C07286=1065.476,339.617,397.493,174.276,33.867,156.261
C07287=1065.483,339.864,397.457,174.280,33.872,156.262
C07288=1065.489,340.112,397.422,174.283,33.877,156.263
C07289=1065.496,340.359,397.387,174.287,33.882,156.264
C07290=1065.501,340.606,397.351,174.291,33.887,156.265
C07291=1065.508,340.853,397.316,174.295,33.893,156.266
C07292=1065.515,341.101,397.281,174.298,33.897,156.267
C07293=1065.521,341.348,397.245,174.302,33.902,156.268
C07294=1065.528,341.596,397.210,174.305,33.908,156.269
C07295=1065.535,341.843,397.175,174.310,33.912,156.270
C07296=1065.541,342.091,397.139,174.313,33.918,156.271
C07297=1065.547,342.338,397.104,174.317,33.923,156.272
C07298=1065.554,342.585,397.069,174.320,33.928,156.273
C07299=1065.560,342.833,397.033,174.324,33.933,156.274
C07300=1065.567,343.081,396.998,174.328,33.938,156.275
C07301=1065.574,343.327,396.962,174.332,33.943,156.276
C07302=1065.581,343.576,396.926,174.336,33.949,156.278
C07303=1065.587,343.823,396.891,174.339,33.954,156.279
C07304=1065.593,344.071,396.855,174.343,33.959,156.280
C07305=1065.601,344.317,396.820,174.347,33.964,156.281
C07306=1065.607,344.565,396.784,174.351,33.969,156.282
C07307=1065.612,344.796,396.751,174.354,33.974,156.283
C07308=1065.618,345.028,396.717,174.358,33.979,156.284
C07309=1065.625,345.260,396.684,174.361,33.984,156.285
C07310=1065.631,345.491,396.650,174.364,33.989,156.286
C07311=1065.637,345.724,396.617,174.369,33.994,156.287
C07312=1065.644,345.955,396.583,174.372,33.998,156.288
C07313=1065.649,346.186,396.550,174.375,34.004,156.289
C07314=1065.655,346.418,396.516,174.379,34.008,156.290
C07315=1065.661,346.665,396.480,174.383,34.013,156.291
C07316=1065.668,346.912,396.444,174.387,34.019,156.292
C07317=1065.675,347.161,396.409,174.390,34.024,156.293
C07318=1065.682,347.408,396.372,174.394,34.029,156.294
C07319=1065.689,347.654,396.336,174.398,34.035,156.296
C07320=1065.695,347.902,396.301,174.402,34.040,156.297
C07321=1065.701,348.149,396.264,174.406,34.045,156.298
C07322=1065.708,348.396,396.229,174.409,34.051,156.299
C07323=1065.714,348.643,396.192,174.413,34.056,156.300
C07324=1065.721,348.891,396.156,174.418,34.062,156.301
C07325=1065.727,349.139,396.120,174.421,34.067,156.302
C07326=1065.734,349.386,396.084,174.425,34.072,156.303
C07327=1065.740,349.633,396.048,174.429,34.077,156.304
C07328=1065.747,349.881,396.012,174.433,34.083,156.306
C07329=1065.754,350.128,395.976,174.437,34.088,156.307
C07330=1065.760,350.375,395.939,174.441,34.093,156.308
C07331=1065.767,350.622,395.903,174.444,34.099,156.309
C07332=1065.774,350.870,395.866,174.448,34.104,156.310
C07333=1065.781,351.117,395.831,174.453,34.110,156.311
C07334=1065.787,351.364,395.794,174.456,34.115,156.312
C07335=1065.793,351.611,395.758,174.460,34.121,156.314
C07336=1065.800,351.859,395.721,174.464,34.126,156.315
C07337=1065.807,352.106,395.685,174.468,34.131,156.316
C07338=1065.814,352.353,395.649,174.472,34.137,156.317
C07339=1065.820,352.600,395.612,174.476,34.142,156.318
C07340=1065.827,352.848,395.576,174.479,34.148,156.319
C07341=1065.833,353.095,395.539,174.484,34.153,156.321
C07342=1065.840,353.342,395.502,174.488,34.159,156.322
C07343=1065.846,353.589,395.466,174.491,34.164,156.323
C07344=1065.853,353.836,395.429,174.496,34.170,156.324
C07345=1065.860,354.084,395.393,174.500,34.175,156.325
C07346=1065.866,354.331,395.356,174.503,34.181,156.326
C07347=1065.872,354.578,395.320,174.507,34.187,156.328
C07348=1065.880,354.825,395.282,174.512,34.192,156.329
C07349=1065.886,355.072,395.246,174.516,34.198,156.330
C07350=1065.892,355.320,395.209,174.519,34.203,156.331
C07351=1065.899,355.567,395.173,174.523,34.209,156.332
C07352=1065.906,355.814,395.136,174.528,34.214,156.333
C07353=1065.913,356.061,395.099,174.532,34.220,156.335
C07354=1065.919,356.309,395.062,174.535,34.226,156.336
C07355=1065.926,356.556,395.025,174.540,34.232,156.337
C07356=1065.933,356.803,394.988,174.544,34.237,156.338
C07357=1065.939,357.050,394.952,174.548,34.243,156.339
C07358=1065.946,357.298,394.915,174.551,34.248,156.341
C07359=1065.953,357.544,394.878,174.556,34.254,156.342
C07360=1065.960,357.792,394.841,174.560,34.260,156.343
C07361=1065.966,358.038,394.804,174.564,34.265,156.344
C07362=1065.973,358.286,394.767,174.568,34.271,156.346
C07363=1065.979,358.520,394.732,174.572,34.276,156.347
C07364=1065.986,358.753,394.697,174.576,34.281,156.348
C07365=1065.992,358.987,394.662,174.579,34.287,156.349
C07366=1065.999,359.221,394.626,174.584,34.292,156.350
C07367=1066.005,359.454,394.591,174.587,34.298,156.351
C07368=1066.011,359.688,394.556,174.591,34.303,156.352
C07369=1066.017,359.922,394.521,174.596,34.309,156.354
C07370=1066.024,360.155,394.486,174.599,34.315,156.355
C07371=1066.030,360.402,394.449,174.603,34.320,156.356
C07372=1066.038,360.649,394.412,174.608,34.326,156.357
C07373=1066.044,360.896,394.374,174.612,34.332,156.359
C07374=1066.051,361.143,394.338,174.615,34.337,156.360
C07375=1066.058,361.391,394.300,174.620,34.343,156.361
C07376=1066.064,361.637,394.262,174.624,34.349,156.362
C07377=1066.071,361.885,394.225,174.628,34.355,156.364
C07378=1066.078,362.132,394.188,174.632,34.361,156.365
C07379=1066.084,362.379,394.150,174.637,34.367,156.366
C07380=1066.092,362.626,394.113,174.641,34.373,156.367
C07381=1066.098,362.873,394.076,174.644,34.379,156.369
C07382=1066.105,363.120,394.037,174.649,34.385,156.370
C07383=1066.112,363.367,394.000,174.653,34.391,156.371
C07384=1066.119,363.614,393.963,174.657,34.396,156.373
C07385=1066.126,363.861,393.925,174.662,34.403,156.374
C07386=1066.132,364.108,393.887,174.666,34.408,156.375
C07387=1066.139,364.355,393.850,174.671,34.414,156.377
C07388=1066.146,364.602,393.812,174.675,34.420,156.378
C07389=1066.153,364.849,393.774,174.678,34.426,156.379
C07390=1066.159,365.097,393.736,174.683,34.432,156.380
C07391=1066.166,365.343,393.699,174.687,34.438,156.382
C07392=1066.172,365.591,393.661,174.691,34.445,156.383
C07393=1066.180,365.838,393.623,174.696,34.451,156.384
C07394=1066.186,366.084,393.586,174.700,34.457,156.386
C07395=1066.193,366.331,393.547,174.704,34.463,156.387
C07396=1066.200,366.578,393.509,174.709,34.469,156.388
C07397=1066.207,366.825,393.472,174.713,34.475,156.390
C07398=1066.213,367.072,393.434,174.718,34.481,156.391
C07399=1066.220,367.319,393.396,174.722,34.487,156.392
C07400=1066.227,367.566,393.358,174.725,34.493,156.394
C07401=1066.233,367.814,393.320,174.730,34.500,156.395
C07402=1066.241,368.060,393.281,174.734,34.506,156.396
C07403=1066.247,368.307,393.244,174.738,34.512,156.398
C07404=1066.254,368.554,393.206,174.743,34.518,156.399
C07405=1066.261,368.801,393.167,174.747,34.524,156.400
C07406=1066.267,369.048,393.129,174.752,34.530,156.402
C07407=1066.275,369.295,393.091,174.756,34.536,156.403
C07408=1066.281,369.542,393.053,174.760,34.543,156.404
C07409=1066.289,369.789,393.014,174.765,34.549,156.406
C07410=1066.295,370.036,392.977,174.769,34.555,156.407
C07411=1066.302,370.282,392.938,174.774,34.562,156.409
C07412=1066.309,370.529,392.900,174.778,34.568,156.410
C07413=1066.316,370.776,392.861,174.782,34.574,156.411
C07414=1066.323,371.023,392.823,174.787,34.581,156.413
C07415=1066.330,371.270,392.785,174.791,34.587,156.414
C07416=1066.337,371.517,392.746,174.796,34.593,156.416
C07417=1066.344,371.764,392.708,174.800,34.599,156.417
C07418=1066.351,372.011,392.670,174.805,34.606,156.418
C07419=1066.358,372.254,392.632,174.809,34.612,156.420
C07420=1066.364,372.496,392.594,174.813,34.618,156.421
C07421=1066.371,372.737,392.556,174.818,34.625,156.423
C07422=1066.378,372.980,392.518,174.822,34.631,156.424
C07423=1066.385,373.222,392.480,174.827,34.637,156.425
C07424=1066.392,373.465,392.442,174.831,34.644,156.427
C07425=1066.398,373.707,392.405,174.836,34.650,156.428
C07426=1066.405,373.950,392.367,174.840,34.656,156.430
C07427=1066.412,374.197,392.328,174.844,34.663,156.431
C07428=1066.419,374.444,392.289,174.849,34.669,156.432
C07429=1066.426,374.690,392.250,174.853,34.676,156.434
C07430=1066.433,374.937,392.211,174.858,34.683,156.435
C07431=1066.439,375.184,392.173,174.862,34.689,156.437
C07432=1066.447,375.430,392.133,174.867,34.695,156.438
C07433=1066.453,375.677,392.094,174.872,34.702,156.440
C07434=1066.460,375.924,392.055,174.877,34.708,156.441
C07435=1066.467,376.171,392.017,174.881,34.715,156.443
C07436=1066.474,376.418,391.978,174.886,34.722,156.444
C07437=1066.481,376.664,391.939,174.890,34.729,156.446
C07438=1066.487,376.911,391.900,174.895,34.735,156.447
C07439=1066.495,377.158,391.860,174.899,34.742,156.449
C07440=1066.502,377.405,391.821,174.903,34.748,156.450
C07441=1066.509,377.652,391.782,174.908,34.755,156.452
C07442=1066.516,377.899,391.744,174.913,34.762,156.453
C07443=1066.523,378.145,391.704,174.918,34.768,156.455
C07444=1066.530,378.392,391.665,174.922,34.775,156.456
C07445=1066.537,378.639,391.625,174.927,34.782,156.458
C07446=1066.544,378.885,391.586,174.931,34.789,156.459
C07447=1066.551,379.132,391.548,174.936,34.795,156.461
C07448=1066.558,379.378,391.508,174.941,34.802,156.462
C07449=1066.565,379.626,391.469,174.946,34.809,156.464
C07450=1066.573,379.872,391.429,174.950,34.816,156.465
C07451=1066.579,380.119,391.391,174.955,34.823,156.467
C07452=1066.587,380.366,391.351,174.960,34.829,156.468
C07453=1066.594,380.613,391.312,174.965,34.836,156.470
C07454=1066.601,380.859,391.272,174.970,34.843,156.471
C07455=1066.609,381.106,391.232,174.974,34.850,156.473
C07456=1066.616,381.353,391.193,174.979,34.857,156.474
C07457=1066.622,381.599,391.153,174.983,34.864,156.476
C07458=1066.630,381.846,391.113,174.989,34.871,156.478
C07459=1066.636,382.093,391.075,174.993,34.878,156.479
C07460=1066.643,382.339,391.034,174.998,34.885,156.481
C07461=1066.651,382.586,390.994,175.002,34.892,156.482
C07462=1066.658,382.832,390.955,175.008,34.899,156.484
C07463=1066.664,383.079,390.915,175.012,34.906,156.485
C07464=1066.672,383.326,390.875,175.017,34.913,156.487
C07465=1066.679,383.573,390.836,175.022,34.920,156.489
C07466=1066.685,383.819,390.796,175.027,34.928,156.490
C07467=1066.693,384.066,390.756,175.032,34.934,156.492
C07468=1066.700,384.312,390.716,175.036,34.941,156.494
C07469=1066.707,384.560,390.676,175.041,34.949,156.495
C07470=1066.714,384.806,390.636,175.047,34.956,156.497
C07471=1066.720,385.052,390.596,175.051,34.963,156.498
C07472=1066.728,385.299,390.556,175.056,34.970,156.500
C07473=1066.735,385.545,390.516,175.061,34.978,156.502
C07474=1066.742,385.792,390.475,175.066,34.985,156.503
C07475=1066.750,386.060,390.432,175.072,34.993,156.505
C07476=1066.758,386.328,390.389,175.076,35.000,156.507
C07477=1066.766,386.596,390.345,175.082,35.008,156.509
C07478=1066.774,386.865,390.302,175.088,35.016,156.510
C07479=1066.782,387.111,390.261,175.092,35.024,156.512
C07480=1066.788,387.357,390.221,175.097,35.031,156.514
C07481=1066.796,387.604,390.181,175.102,35.038,156.516
C07482=1066.802,387.851,390.141,175.107,35.045,156.517
C07483=1066.810,388.097,390.100,175.113,35.052,156.519
C07484=1066.817,388.344,390.060,175.117,35.060,156.521
C07485=1066.825,388.590,390.019,175.122,35.067,156.522
C07486=1066.832,388.837,389.979,175.128,35.075,156.524
C07487=1066.840,389.083,389.938,175.132,35.082,156.526
C07488=1066.847,389.330,389.899,175.137,35.089,156.527
C07489=1066.854,389.576,389.857,175.143,35.097,156.529
C07490=1066.862,389.823,389.817,175.147,35.104,156.531
C07491=1066.868,390.069,389.777,175.153,35.112,156.533
C07492=1066.876,390.316,389.737,175.157,35.119,156.534
C07493=1066.884,390.563,389.695,175.163,35.127,156.536
C07494=1066.890,390.810,389.655,175.168,35.134,156.538
C07495=1066.898,391.055,389.615,175.174,35.142,156.539
C07496=1066.905,391.302,389.573,175.178,35.150,156.541
C07497=1066.912,391.549,389.532,175.183,35.157,156.543
C07498=1066.920,391.795,389.492,175.189,35.165,156.545
C07499=1066.927,392.041,389.451,175.193,35.173,156.547
C07500=1066.934,392.288,389.410,175.199,35.181,156.548
C07501=1066.942,392.534,389.370,175.204,35.188,156.550
C07502=1066.949,392.781,389.328,175.209,35.196,156.552
C07503=1066.956,393.027,389.287,175.214,35.204,156.554
C07504=1066.963,393.273,389.246,175.220,35.211,156.556
C07505=1066.971,393.520,389.206,175.225,35.219,156.557
C07506=1066.979,393.766,389.164,175.230,35.227,156.559
C07507=1066.986,394.013,389.123,175.235,35.234,156.561
C07508=1066.993,394.259,389.082,175.241,35.243,156.563
C07509=1067.000,394.505,389.041,175.246,35.250,156.565
C07510=1067.007,394.752,389.000,175.251,35.258,156.566
C07511=1067.015,394.998,388.959,175.256,35.266,156.568
C07512=1067.023,395.245,388.918,175.262,35.274,156.570
C07513=1067.030,395.491,388.877,175.267,35.282,156.572
C07514=1067.038,395.737,388.835,175.272,35.290,156.574
C07515=1067.045,395.984,388.794,175.278,35.298,156.576
C07516=1067.052,396.230,388.752,175.283,35.306,156.578
C07517=1067.059,396.477,388.711,175.289,35.314,156.579
C07518=1067.067,396.723,388.669,175.293,35.322,156.581
C07519=1067.074,396.970,388.628,175.299,35.330,156.583
C07520=1067.082,397.216,388.587,175.304,35.338,156.585
C07521=1067.089,397.462,388.545,175.310,35.346,156.587
C07522=1067.096,397.709,388.503,175.316,35.354,156.589
C07523=1067.104,397.955,388.462,175.320,35.362,156.591
C07524=1067.111,398.201,388.420,175.326,35.370,156.593
C07525=1067.119,398.447,388.378,175.332,35.379,156.595
C07526=1067.127,398.695,388.337,175.337,35.387,156.597
C07527=1067.134,398.941,388.295,175.343,35.395,156.598
C07528=1067.142,399.187,388.254,175.348,35.403,156.600
C07529=1067.149,399.433,388.211,175.353,35.412,156.602
C07530=1067.156,399.679,388.169,175.359,35.420,156.604
C07531=1067.165,399.963,388.121,175.365,35.429,156.607
C07532=1067.174,400.249,388.073,175.372,35.439,156.609
C07533=1067.182,400.533,388.025,175.378,35.449,156.611
C07534=1067.191,400.817,387.976,175.384,35.459,156.614
C07535=1067.198,401.064,387.933,175.390,35.467,156.615
C07536=1067.206,401.310,387.891,175.396,35.475,156.617
C07537=1067.214,401.556,387.850,175.401,35.484,156.619
C07538=1067.221,401.802,387.808,175.407,35.492,156.621
C07539=1067.229,402.048,387.765,175.413,35.501,156.623
C07540=1067.236,402.295,387.723,175.419,35.509,156.625
C07541=1067.244,402.541,387.681,175.423,35.517,156.627
C07542=1067.252,402.787,387.638,175.429,35.526,156.630
C07543=1067.260,403.033,387.597,175.435,35.535,156.632
C07544=1067.266,403.279,387.554,175.441,35.544,156.634
C07545=1067.275,403.526,387.512,175.446,35.552,156.636
C07546=1067.282,403.772,387.470,175.452,35.561,156.638
C07547=1067.290,404.019,387.427,175.458,35.570,156.640
C07548=1067.297,404.265,387.385,175.464,35.578,156.642
C07549=1067.304,404.511,387.342,175.470,35.587,156.644
C07550=1067.313,404.757,387.299,175.475,35.596,156.646
C07551=1067.320,405.003,387.257,175.481,35.604,156.648
C07552=1067.328,405.250,387.214,175.487,35.613,156.650
C07553=1067.336,405.496,387.172,175.493,35.622,156.652
C07554=1067.343,405.743,387.129,175.499,35.631,156.655
C07555=1067.351,405.988,387.086,175.505,35.640,156.657
C07556=1067.358,406.235,387.043,175.511,35.649,156.659
C07557=1067.366,406.480,387.001,175.516,35.657,156.661
C07558=1067.374,406.727,386.958,175.522,35.666,156.663
C07559=1067.381,406.973,386.915,175.528,35.676,156.665
C07560=1067.389,407.220,386.872,175.534,35.684,156.667
C07561=1067.396,407.465,386.829,175.540,35.694,156.670
C07562=1067.404,407.712,386.785,175.546,35.703,156.672
C07563=1067.412,407.958,386.743,175.552,35.712,156.674
C07564=1067.419,408.204,386.700,175.558,35.721,156.676
C07565=1067.427,408.450,386.656,175.564,35.730,156.678
C07566=1067.435,408.696,386.614,175.570,35.739,156.681
C07567=1067.443,408.943,386.571,175.576,35.749,156.683
C07568=1067.450,409.189,386.527,175.582,35.758,156.685
C07569=1067.458,409.435,386.484,175.588,35.767,156.687
C07570=1067.466,409.681,386.441,175.595,35.776,156.690
C07571=1067.474,409.927,386.397,175.601,35.785,156.692
C07572=1067.482,410.173,386.354,175.607,35.795,156.694
C07573=1067.489,410.419,386.311,175.613,35.804,156.696
C07574=1067.497,410.665,386.267,175.619,35.813,156.699
C07575=1067.505,410.912,386.224,175.625,35.823,156.701
C07576=1067.513,411.158,386.181,175.631,35.832,156.703
C07577=1067.521,411.403,386.137,175.637,35.842,156.705
C07578=1067.528,411.650,386.094,175.643,35.851,156.708
C07579=1067.537,411.896,386.051,175.650,35.860,156.710
C07580=1067.545,412.142,386.006,175.656,35.870,156.712
C07581=1067.553,412.388,385.963,175.662,35.879,156.715
C07582=1067.560,412.634,385.919,175.668,35.889,156.717
C07583=1067.569,412.880,385.876,175.674,35.898,156.719
C07584=1067.577,413.126,385.832,175.682,35.908,156.722
C07585=1067.585,413.373,385.788,175.688,35.918,156.724
C07586=1067.593,413.618,385.744,175.694,35.927,156.726
C07587=1067.601,413.907,385.693,175.701,35.939,156.729
C07588=1067.612,414.195,385.642,175.709,35.950,156.732
C07589=1067.621,414.484,385.590,175.716,35.961,156.735
C07590=1067.630,414.772,385.539,175.724,35.973,156.738
C07591=1067.638,415.018,385.494,175.731,35.982,156.740
C07592=1067.646,415.265,385.451,175.737,35.993,156.742
C07593=1067.654,415.510,385.406,175.743,36.002,156.745
C07594=1067.662,415.756,385.362,175.750,36.012,156.747
C07595=1067.670,416.002,385.318,175.756,36.022,156.750
C07596=1067.678,416.248,385.274,175.763,36.032,156.752
C07597=1067.686,416.494,385.230,175.770,36.042,156.755
C07598=1067.694,416.740,385.185,175.776,36.052,156.757
C07599=1067.703,416.986,385.141,175.783,36.062,156.760
C07600=1067.710,417.232,385.096,175.790,36.073,156.762
C07601=1067.718,417.478,385.051,175.796,36.083,156.765
C07602=1067.726,417.724,385.007,175.803,36.093,156.767
C07603=1067.734,417.969,384.963,175.810,36.103,156.770
C07604=1067.742,418.215,384.918,175.816,36.113,156.772
C07605=1067.751,418.462,384.874,175.823,36.123,156.775
C07606=1067.759,418.707,384.829,175.830,36.134,156.777
C07607=1067.767,418.953,384.785,175.836,36.144,156.780
C07608=1067.775,419.198,384.739,175.844,36.154,156.782
C07609=1067.783,419.445,384.695,175.850,36.165,156.785
C07610=1067.791,419.691,384.650,175.857,36.175,156.788
C07611=1067.800,419.936,384.606,175.864,36.185,156.790
C07612=1067.808,420.182,384.561,175.870,36.196,156.793
C07613=1067.817,420.428,384.516,175.878,36.206,156.795
C07614=1067.824,420.673,384.470,175.884,36.217,156.798
C07615=1067.833,420.920,384.426,175.892,36.227,156.801
C07616=1067.841,421.165,384.381,175.898,36.238,156.803
C07617=1067.849,421.411,384.336,175.906,36.248,156.806
C07618=1067.858,421.657,384.290,175.912,36.259,156.809
C07619=1067.865,421.903,384.245,175.920,36.270,156.811
C07620=1067.874,422.149,384.200,175.926,36.281,156.814
C07621=1067.882,422.394,384.155,175.934,36.291,156.817
C07622=1067.890,422.639,384.109,175.941,36.302,156.819
C07623=1067.899,422.886,384.065,175.948,36.313,156.822
C07624=1067.906,423.131,384.019,175.955,36.323,156.825
C07625=1067.915,423.377,383.974,175.962,36.335,156.828
C07626=1067.923,423.622,383.928,175.969,36.345,156.830
C07627=1067.932,423.868,383.882,175.977,36.356,156.833
C07628=1067.939,424.114,383.837,175.983,36.367,156.836
C07629=1067.948,424.360,383.791,175.991,36.378,156.839
C07630=1067.957,424.606,383.745,175.998,36.389,156.842
C07631=1067.965,424.851,383.700,176.005,36.400,156.844
C07632=1067.973,425.097,383.654,176.013,36.411,156.847
C07633=1067.982,425.342,383.609,176.021,36.423,156.850
C07634=1067.990,425.588,383.563,176.027,36.434,156.853
C07635=1067.999,425.833,383.517,176.035,36.445,156.856
C07636=1068.007,426.079,383.471,176.043,36.456,156.858
C07637=1068.016,426.325,383.426,176.049,36.467,156.861
C07638=1068.024,426.571,383.380,176.057,36.478,156.864
C07639=1068.033,426.816,383.334,176.065,36.490,156.867
C07640=1068.042,427.062,383.288,176.072,36.501,156.870
C07641=1068.050,427.307,383.242,176.080,36.512,156.873
C07642=1068.058,427.553,383.196,176.087,36.524,156.876
C07643=1068.068,427.821,383.145,176.096,36.536,156.879
C07644=1068.077,428.089,383.095,176.104,36.549,156.882
C07645=1068.086,428.358,383.044,176.113,36.562,156.885
C07646=1068.095,428.626,382.994,176.121,36.574,156.889
C07647=1068.105,428.912,382.940,176.130,36.588,156.892
C07648=1068.115,429.196,382.886,176.139,36.601,156.896
C07649=1068.125,429.481,382.832,176.147,36.615,156.899
C07650=1068.135,429.766,382.778,176.156,36.629,156.903
C07651=1068.145,430.011,382.732,176.164,36.640,156.906
C07652=1068.153,430.257,382.685,176.172,36.652,156.909
C07653=1068.162,430.503,382.638,176.180,36.664,156.912
C07654=1068.170,430.748,382.591,176.188,36.676,156.915
C07655=1068.179,430.994,382.545,176.196,36.688,156.918
C07656=1068.188,431.239,382.499,176.203,36.700,156.921
C07657=1068.197,431.484,382.452,176.211,36.712,156.924
C07658=1068.205,431.730,382.405,176.219,36.723,156.927
C07659=1068.214,431.975,382.358,176.227,36.736,156.931
C07660=1068.223,432.220,382.311,176.235,36.748,156.934
C07661=1068.231,432.466,382.264,176.243,36.760,156.937
C07662=1068.239,432.711,382.216,176.252,36.772,156.940
C07663=1068.248,432.956,382.169,176.260,36.785,156.943
C07664=1068.256,433.202,382.123,176.268,36.797,156.946
C07665=1068.265,433.447,382.075,176.276,36.809,156.950
C07666=1068.275,433.692,382.027,176.285,36.822,156.953
C07667=1068.283,433.938,381.981,176.293,36.834,156.956
C07668=1068.292,434.183,381.933,176.301,36.847,156.959
C07669=1068.301,434.428,381.886,176.310,36.859,156.963
C07670=1068.309,434.673,381.839,176.318,36.872,156.966
C07671=1068.319,434.919,381.791,176.326,36.884,156.969
C07672=1068.328,435.164,381.744,176.334,36.897,156.973
C07673=1068.337,435.409,381.696,176.343,36.909,156.976
C07674=1068.345,435.655,381.648,176.351,36.922,156.979
C07675=1068.354,435.899,381.601,176.360,36.935,156.983
C07676=1068.363,436.144,381.553,176.368,36.948,156.986
C07677=1068.372,436.390,381.505,176.377,36.960,156.989
C07678=1068.381,436.635,381.458,176.385,36.973,156.993
C07679=1068.391,436.880,381.410,176.394,36.986,156.996
C07680=1068.400,437.125,381.363,176.403,36.999,156.999
C07681=1068.408,437.371,381.314,176.411,37.012,157.003
C07682=1068.417,437.616,381.267,176.420,37.024,157.006
C07683=1068.427,437.861,381.218,176.429,37.038,157.010
C07684=1068.436,438.106,381.171,176.437,37.051,157.013
C07685=1068.445,438.352,381.123,176.446,37.064,157.017
C07686=1068.454,438.597,381.074,176.455,37.077,157.020
C07687=1068.463,438.842,381.026,176.464,37.090,157.024
C07688=1068.473,439.087,380.978,176.472,37.103,157.027
C07689=1068.481,439.332,380.930,176.482,37.117,157.031
C07690=1068.491,439.577,380.881,176.490,37.130,157.034
C07691=1068.500,439.822,380.832,176.500,37.143,157.038
C07692=1068.509,440.067,380.785,176.508,37.157,157.042
C07693=1068.518,440.312,380.736,176.518,37.171,157.045
C07694=1068.527,440.557,380.687,176.527,37.184,157.049
C07695=1068.537,440.802,380.639,176.536,37.198,157.052
C07696=1068.546,441.047,380.590,176.545,37.211,157.056
C07697=1068.555,441.292,380.541,176.554,37.225,157.060
C07698=1068.564,441.537,380.492,176.563,37.239,157.063
C07699=1068.578,441.892,380.422,176.577,37.259,157.069
C07700=1068.591,442.245,380.351,176.590,37.279,157.074
C07701=1068.605,442.599,380.281,176.604,37.299,157.080
C07702=1068.619,442.953,380.210,176.618,37.319,157.085
C07703=1068.628,443.199,380.161,176.627,37.333,157.089
C07704=1068.637,443.443,380.111,176.637,37.347,157.093
C07705=1068.647,443.688,380.062,176.646,37.361,157.096
C07706=1068.656,443.933,380.012,176.655,37.375,157.100
C07707=1068.665,444.178,379.963,176.665,37.389,157.104
C07708=1068.675,444.422,379.914,176.675,37.404,157.108
C07709=1068.684,444.668,379.865,176.685,37.418,157.112
C07710=1068.693,444.912,379.815,176.695,37.432,157.116
C07711=1068.704,445.157,379.766,176.705,37.447,157.120
C07712=1068.713,445.401,379.716,176.714,37.461,157.124
C07713=1068.722,445.646,379.666,176.724,37.476,157.128
C07714=1068.731,445.891,379.617,176.734,37.490,157.132
C07715=1068.741,446.136,379.568,176.744,37.505,157.136
C07716=1068.751,446.381,379.518,176.754,37.519,157.140
C07717=1068.761,446.626,379.468,176.764,37.534,157.144
C07718=1068.770,446.870,379.417,176.774,37.549,157.148
C07719=1068.780,447.114,379.367,176.784,37.563,157.152
C07720=1068.790,447.359,379.318,176.794,37.579,157.156
C07721=1068.800,447.604,379.268,176.804,37.593,157.160
C07722=1068.809,447.849,379.218,176.814,37.608,157.164
C07723=1068.819,448.093,379.168,176.824,37.623,157.168
C07724=1068.830,448.335,379.119,176.835,37.638,157.172
C07725=1068.841,448.580,379.070,176.844,37.652,157.176
C07726=1068.855,448.825,379.022,176.854,37.666,157.180
C07727=1068.869,449.070,378.975,176.864,37.679,157.184
C07728=1068.884,449.315,378.928,176.873,37.692,157.188
C07729=1068.900,449.560,378.882,176.881,37.705,157.191
C07730=1068.918,449.806,378.837,176.890,37.717,157.194
C07731=1068.572,449.808,378.581,176.879,37.852,157.231
C07732=1068.554,449.562,378.625,176.870,37.840,157.227
C07733=1068.538,449.317,378.671,176.860,37.827,157.224
C07734=1068.523,449.071,378.718,176.851,37.814,157.220
C07735=1068.509,448.827,378.765,176.842,37.801,157.216
C07736=1068.495,448.582,378.814,176.832,37.787,157.213
C07737=1068.483,448.337,378.862,176.822,37.773,157.209
C07738=1068.472,448.094,378.911,176.812,37.759,157.205
C07739=1068.462,447.851,378.961,176.801,37.743,157.200
C07740=1068.453,447.606,379.011,176.790,37.729,157.196
C07741=1068.443,447.361,379.061,176.780,37.714,157.192
C07742=1068.433,447.117,379.112,176.770,37.699,157.188
C07743=1068.423,446.872,379.161,176.760,37.684,157.184
C07744=1068.413,446.627,379.211,176.750,37.670,157.180
C07745=1068.404,446.382,379.261,176.740,37.655,157.176
C07746=1068.395,446.138,379.311,176.730,37.640,157.172
C07747=1068.385,445.892,379.361,176.720,37.625,157.168
C07748=1068.375,445.648,379.410,176.710,37.611,157.164
C07749=1068.365,445.403,379.460,176.700,37.597,157.160
C07750=1068.356,445.159,379.510,176.690,37.582,157.156
C07751=1068.346,444.914,379.559,176.680,37.568,157.152
C07752=1068.336,444.670,379.609,176.670,37.553,157.148
C07753=1068.327,444.424,379.658,176.660,37.539,157.144
C07754=1068.318,444.180,379.708,176.650,37.525,157.140
C07755=1068.308,443.935,379.757,176.640,37.511,157.136
C07756=1068.298,443.689,379.807,176.631,37.496,157.132
C07757=1068.289,443.445,379.856,176.622,37.483,157.129
C07758=1068.279,443.200,379.905,176.612,37.468,157.125
C07759=1068.270,442.955,379.954,176.602,37.455,157.121
C07760=1068.257,442.620,380.021,176.589,37.435,157.116
C07761=1068.244,442.285,380.088,176.576,37.416,157.111
C07762=1068.232,441.949,380.155,176.563,37.398,157.105
C07763=1068.219,441.614,380.223,176.550,37.379,157.100
C07764=1068.209,441.369,380.271,176.541,37.365,157.097
C07765=1068.200,441.124,380.320,176.532,37.352,157.093
C07766=1068.191,440.880,380.368,176.523,37.338,157.089
C07767=1068.182,440.635,380.418,176.513,37.324,157.086
C07768=1068.172,440.390,380.466,176.504,37.311,157.082
C07769=1068.163,440.144,380.515,176.495,37.297,157.078
C07770=1068.154,439.900,380.563,176.486,37.284,157.075
C07771=1068.145,439.654,380.611,176.477,37.271,157.071
C07772=1068.136,439.409,380.660,176.467,37.257,157.068
C07773=1068.127,439.165,380.708,176.459,37.244,157.064
C07774=1068.118,438.919,380.757,176.449,37.231,157.060
C07775=1068.108,438.674,380.805,176.441,37.218,157.057
C07776=1068.099,438.430,380.854,176.431,37.204,157.053
C07777=1068.090,438.184,380.902,176.423,37.191,157.050
C07778=1068.081,437.939,380.949,176.415,37.178,157.046
C07779=1068.072,437.694,380.998,176.405,37.165,157.043
C07780=1068.062,437.448,381.046,176.397,37.152,157.040
C07781=1068.053,437.204,381.093,176.388,37.139,157.036
C07782=1068.044,436.959,381.142,176.379,37.127,157.033
C07783=1068.035,436.713,381.190,176.371,37.114,157.029
C07784=1068.026,436.468,381.238,176.362,37.101,157.026
C07785=1068.017,436.223,381.285,176.353,37.088,157.022
C07786=1068.008,435.977,381.333,176.345,37.075,157.019
C07787=1067.999,435.732,381.380,176.336,37.063,157.016
C07788=1067.990,435.488,381.428,176.328,37.050,157.012
C07789=1067.980,435.242,381.475,176.319,37.037,157.009
C07790=1067.972,434.997,381.523,176.310,37.025,157.006
C07791=1067.964,434.752,381.571,176.302,37.012,157.002
C07792=1067.954,434.506,381.619,176.294,36.999,156.999
C07793=1067.946,434.261,381.666,176.285,36.987,156.996
C07794=1067.937,434.016,381.713,176.277,36.975,156.992
C07795=1067.928,433.771,381.760,176.268,36.963,156.989
C07796=1067.919,433.525,381.808,176.260,36.950,156.986
C07797=1067.910,433.280,381.855,176.252,36.938,156.983
C07798=1067.901,433.034,381.902,176.244,36.925,156.980
C07799=1067.892,432.789,381.949,176.236,36.913,156.976
C07800=1067.884,432.544,381.996,176.228,36.901,156.973
C07801=1067.875,432.299,382.043,176.220,36.889,156.970
C07802=1067.866,432.054,382.090,176.211,36.876,156.967
C07803=1067.857,431.808,382.138,176.202,36.865,156.964
C07804=1067.848,431.562,382.185,176.194,36.853,156.961
C07805=1067.840,431.317,382.231,176.186,36.841,156.957
C07806=1067.831,431.071,382.278,176.178,36.829,156.954
C07807=1067.823,430.826,382.325,176.170,36.817,156.951
C07808=1067.814,430.581,382.372,176.162,36.805,156.948
C07809=1067.805,430.335,382.419,176.155,36.793,156.945
C07810=1067.797,430.090,382.466,176.147,36.781,156.942
C07811=1067.788,429.845,382.512,176.139,36.769,156.939
C07812=1067.779,429.599,382.559,176.131,36.758,156.936
C07813=1067.771,429.354,382.605,176.124,36.746,156.933
C07814=1067.762,429.108,382.651,176.116,36.734,156.930
C07815=1067.753,428.862,382.697,176.108,36.723,156.927
C07816=1067.743,428.553,382.756,176.098,36.708,156.923
C07817=1067.732,428.243,382.815,176.088,36.693,156.919
C07818=1067.721,427.934,382.873,176.079,36.679,156.915
C07819=1067.710,427.624,382.932,176.069,36.665,156.912
C07820=1067.702,427.379,382.977,176.061,36.653,156.909
C07821=1067.693,427.133,383.024,176.054,36.642,156.906
C07822=1067.685,426.887,383.070,176.046,36.631,156.903
C07823=1067.676,426.641,383.115,176.039,36.619,156.900
C07824=1067.668,426.396,383.162,176.031,36.608,156.897
C07825=1067.659,426.150,383.207,176.023,36.596,156.894
C07826=1067.651,425.905,383.254,176.016,36.585,156.892
C07827=1067.642,425.660,383.299,176.009,36.574,156.889
C07828=1067.633,425.413,383.345,176.001,36.563,156.886
C07829=1067.625,425.168,383.390,175.994,36.552,156.883
C07830=1067.617,424.923,383.437,175.986,36.541,156.880
C07831=1067.608,424.677,383.482,175.979,36.530,156.877
C07832=1067.600,424.431,383.528,175.971,36.519,156.875
C07833=1067.591,424.186,383.573,175.964,36.508,156.872
C07834=1067.583,423.940,383.619,175.957,36.497,156.869
C07835=1067.574,423.694,383.665,175.950,36.486,156.866
C07836=1067.566,423.448,383.711,175.943,36.475,156.864
C07837=1067.558,423.203,383.756,175.935,36.464,156.861
C07838=1067.549,422.957,383.802,175.928,36.454,156.858
C07839=1067.541,422.711,383.846,175.921,36.443,156.855
C07840=1067.532,422.465,383.891,175.914,36.432,156.853
C07841=1067.525,422.220,383.937,175.906,36.421,156.850
C07842=1067.516,421.974,383.982,175.899,36.411,156.847
C07843=1067.508,421.728,384.027,175.892,36.400,156.844
C07844=1067.500,421.483,384.072,175.885,36.389,156.842
C07845=1067.492,421.237,384.118,175.878,36.379,156.839
C07846=1067.484,420.991,384.163,175.871,36.368,156.836
C07847=1067.475,420.745,384.208,175.864,36.358,156.834
C07848=1067.467,420.500,384.253,175.857,36.347,156.831
C07849=1067.459,420.254,384.298,175.850,36.337,156.828
C07850=1067.450,420.008,384.343,175.844,36.326,156.826
C07851=1067.442,419.763,384.388,175.836,36.316,156.823
C07852=1067.435,419.541,384.429,175.830,36.307,156.821
C07853=1067.427,419.319,384.469,175.824,36.297,156.819
C07854=1067.420,419.097,384.509,175.817,36.288,156.816
C07855=1067.412,418.875,384.550,175.812,36.279,156.814
C07856=1067.405,418.653,384.589,175.806,36.270,156.812
C07857=1067.397,418.431,384.629,175.799,36.260,156.809
C07858=1067.390,418.209,384.670,175.793,36.251,156.807
C07859=1067.383,417.988,384.710,175.787,36.242,156.805
C07860=1067.375,417.742,384.755,175.780,36.232,156.802
C07861=1067.367,417.496,384.799,175.773,36.221,156.800
C07862=1067.359,417.250,384.844,175.767,36.212,156.797
C07863=1067.350,417.004,384.888,175.760,36.202,156.795
C07864=1067.342,416.758,384.933,175.754,36.192,156.792
C07865=1067.334,416.512,384.977,175.747,36.181,156.790
C07866=1067.326,416.266,385.021,175.740,36.171,156.787
C07867=1067.318,416.021,385.066,175.734,36.161,156.785
C07868=1067.310,415.775,385.110,175.726,36.152,156.782
C07869=1067.302,415.529,385.154,175.720,36.141,156.780
C07870=1067.295,415.283,385.199,175.714,36.132,156.777
C07871=1067.287,415.037,385.243,175.707,36.122,156.775
C07872=1067.275,414.698,385.303,175.699,36.108,156.772
C07873=1067.265,414.361,385.364,175.689,36.095,156.768
C07874=1067.254,414.022,385.424,175.680,36.082,156.765
C07875=1067.242,413.683,385.484,175.671,36.068,156.762
C07876=1067.234,413.437,385.529,175.665,36.059,156.759
C07877=1067.226,413.191,385.572,175.659,36.049,156.757
C07878=1067.217,412.945,385.616,175.653,36.039,156.755
C07879=1067.210,412.699,385.660,175.646,36.030,156.752
C07880=1067.202,412.453,385.703,175.639,36.021,156.750
C07881=1067.194,412.208,385.747,175.633,36.011,156.748
C07882=1067.186,411.962,385.790,175.627,36.001,156.745
C07883=1067.178,411.715,385.834,175.621,35.992,156.743
C07884=1067.170,411.469,385.878,175.614,35.983,156.741
C07885=1067.163,411.222,385.921,175.608,35.973,156.738
C07886=1067.154,410.977,385.965,175.602,35.964,156.736
C07887=1067.146,410.731,386.009,175.596,35.955,156.734
C07888=1067.139,410.485,386.052,175.590,35.945,156.731
C07889=1067.131,410.239,386.095,175.583,35.936,156.729
C07890=1067.123,409.993,386.138,175.577,35.927,156.727
C07891=1067.115,409.746,386.182,175.571,35.917,156.725
C07892=1067.108,409.501,386.225,175.565,35.908,156.722
C07893=1067.099,409.255,386.268,175.559,35.899,156.720
C07894=1067.092,409.008,386.311,175.553,35.890,156.718
C07895=1067.085,408.762,386.355,175.547,35.880,156.716
C07896=1067.076,408.516,386.398,175.540,35.871,156.714
C07897=1067.068,408.269,386.441,175.534,35.862,156.711
C07898=1067.061,408.024,386.484,175.528,35.853,156.709
C07899=1067.053,407.777,386.527,175.522,35.844,156.707
C07900=1067.045,407.531,386.570,175.516,35.835,156.705
C07901=1067.038,407.285,386.614,175.510,35.826,156.703
C07902=1067.030,407.039,386.657,175.504,35.817,156.700
C07903=1067.023,406.793,386.699,175.498,35.808,156.698
C07904=1067.015,406.546,386.743,175.493,35.799,156.696
C07905=1067.007,406.300,386.785,175.487,35.790,156.694
C07906=1067.000,406.054,386.828,175.481,35.781,156.692
C07907=1066.992,405.808,386.870,175.475,35.772,156.690
C07908=1066.984,405.562,386.914,175.469,35.763,156.687
C07909=1066.977,405.316,386.956,175.463,35.755,156.685
C07910=1066.969,405.069,386.999,175.456,35.746,156.683
C07911=1066.961,404.823,387.041,175.451,35.737,156.681
C07912=1066.953,404.577,387.084,175.445,35.728,156.679
C07913=1066.946,404.330,387.126,175.439,35.720,156.677
C07914=1066.938,404.084,387.169,175.433,35.711,156.675
C07915=1066.931,403.838,387.212,175.428,35.702,156.673
C07916=1066.923,403.591,387.254,175.423,35.694,156.671
C07917=1066.915,403.345,387.296,175.417,35.685,156.669
C07918=1066.908,403.099,387.339,175.411,35.676,156.667
C07919=1066.900,402.853,387.382,175.405,35.668,156.664
C07920=1066.892,402.607,387.424,175.399,35.659,156.662
C07921=1066.885,402.360,387.467,175.394,35.651,156.660
C07922=1066.877,402.114,387.508,175.388,35.642,156.658
C07923=1066.870,401.868,387.550,175.382,35.634,156.656
C07924=1066.861,401.622,387.593,175.377,35.625,156.654
C07925=1066.854,401.375,387.634,175.371,35.617,156.652
C07926=1066.847,401.129,387.676,175.365,35.608,156.650
C07927=1066.840,400.883,387.718,175.359,35.600,156.648
C07928=1066.831,400.596,387.767,175.353,35.590,156.646
C07929=1066.821,400.310,387.816,175.347,35.581,156.644
C07930=1066.813,400.025,387.865,175.340,35.571,156.641
C07931=1066.804,399.739,387.914,175.334,35.562,156.639
C07932=1066.797,399.492,387.955,175.328,35.553,156.637
C07933=1066.789,399.246,387.997,175.322,35.545,156.635
C07934=1066.781,399.000,388.039,175.317,35.536,156.633
C07935=1066.774,398.753,388.081,175.311,35.528,156.631
C07936=1066.767,398.507,388.123,175.305,35.520,156.629
C07937=1066.759,398.261,388.165,175.301,35.512,156.627
C07938=1066.752,398.014,388.206,175.295,35.504,156.626
C07939=1066.744,397.768,388.248,175.290,35.496,156.624
C07940=1066.737,397.522,388.289,175.284,35.487,156.622
C07941=1066.730,397.275,388.331,175.278,35.480,156.620
C07942=1066.722,397.029,388.373,175.273,35.471,156.618
C07943=1066.715,396.783,388.414,175.267,35.463,156.616
C07944=1066.707,396.536,388.456,175.263,35.456,156.614
C07945=1066.699,396.289,388.497,175.257,35.447,156.612
C07946=1066.692,396.043,388.539,175.252,35.439,156.610
C07947=1066.684,395.797,388.580,175.246,35.432,156.609
C07948=1066.676,395.550,388.621,175.240,35.423,156.607
C07949=1066.670,395.304,388.662,175.236,35.416,156.605
C07950=1066.662,395.058,388.703,175.230,35.407,156.603
C07951=1066.655,394.811,388.744,175.225,35.400,156.601
C07952=1066.648,394.565,388.786,175.219,35.392,156.599
C07953=1066.640,394.319,388.828,175.214,35.384,156.597
C07954=1066.633,394.072,388.869,175.209,35.376,156.596
C07955=1066.626,393.826,388.910,175.204,35.368,156.594
C07956=1066.618,393.579,388.951,175.198,35.361,156.592
C07957=1066.610,393.333,388.992,175.193,35.353,156.590
C07958=1066.603,393.086,389.033,175.188,35.345,156.588
C07959=1066.596,392.840,389.074,175.183,35.337,156.586
C07960=1066.589,392.594,389.115,175.177,35.329,156.585
C07961=1066.581,392.347,389.156,175.172,35.322,156.583
C07962=1066.574,392.101,389.197,175.167,35.314,156.581
C07963=1066.567,391.853,389.238,175.162,35.307,156.579
C07964=1066.559,391.608,389.278,175.156,35.299,156.578
C07965=1066.552,391.361,389.319,175.151,35.292,156.576
C07966=1066.545,391.115,389.360,175.147,35.284,156.574
C07967=1066.537,390.868,389.401,175.141,35.276,156.572
C07968=1066.530,390.622,389.441,175.136,35.269,156.571
C07969=1066.523,390.375,389.482,175.130,35.261,156.569
C07970=1066.515,390.129,389.523,175.126,35.254,156.567
C07971=1066.508,389.882,389.564,175.120,35.246,156.565
C07972=1066.501,389.636,389.604,175.115,35.239,156.564
C07973=1066.494,389.389,389.644,175.110,35.231,156.562
C07974=1066.486,389.143,389.685,175.105,35.224,156.560
C07975=1066.479,388.896,389.725,175.100,35.217,156.558
C07976=1066.471,388.650,389.766,175.095,35.209,156.557
C07977=1066.464,388.403,389.806,175.090,35.202,156.555
C07978=1066.456,388.156,389.847,175.085,35.194,156.553
C07979=1066.449,387.910,389.886,175.080,35.187,156.552
C07980=1066.442,387.663,389.927,175.075,35.180,156.550
C07981=1066.435,387.417,389.967,175.069,35.172,156.548
C07982=1066.428,387.170,390.008,175.065,35.165,156.547
C07983=1066.420,386.923,390.048,175.060,35.158,156.545
C07984=1066.413,386.654,390.092,175.054,35.150,156.543
C07985=1066.404,386.385,390.136,175.048,35.142,156.541
C07986=1066.396,386.115,390.179,175.043,35.134,156.540
C07987=1066.389,385.845,390.224,175.038,35.126,156.538
C07988=1066.381,385.599,390.263,175.032,35.119,156.536
C07989=1066.375,385.351,390.304,175.028,35.112,156.534
C07990=1066.367,385.105,390.343,175.023,35.105,156.533
C07991=1066.360,384.858,390.383,175.019,35.097,156.531
C07992=1066.353,384.613,390.424,175.013,35.090,156.530
C07993=1066.345,384.366,390.464,175.008,35.084,156.528
C07994=1066.339,384.119,390.504,175.004,35.076,156.526
C07995=1066.332,383.873,390.544,174.998,35.069,156.525
C07996=1066.324,383.626,390.584,174.993,35.062,156.523
C07997=1066.318,383.379,390.623,174.989,35.055,156.521
C07998=1066.310,383.132,390.663,174.984,35.048,156.520
C07999=1066.303,382.886,390.703,174.979,35.041,156.518
C08000=1066.297,382.639,390.743,174.974,35.034,156.517
C08001=1066.289,382.392,390.783,174.969,35.027,156.515
C08002=1066.282,382.146,390.822,174.965,35.020,156.513
C08003=1066.276,381.900,390.862,174.960,35.013,156.512
C08004=1066.268,381.652,390.902,174.955,35.006,156.510
C08005=1066.261,381.406,390.941,174.950,34.999,156.509
C08006=1066.255,381.159,390.981,174.946,34.992,156.507
C08007=1066.247,380.912,391.021,174.941,34.985,156.506
C08008=1066.240,380.666,391.060,174.936,34.978,156.504
C08009=1066.232,380.419,391.100,174.931,34.971,156.502
C08010=1066.226,380.172,391.139,174.926,34.964,156.501
C08011=1066.218,379.926,391.178,174.922,34.958,156.499
C08012=1066.212,379.679,391.217,174.917,34.951,156.498
C08013=1066.204,379.432,391.257,174.913,34.944,156.496
C08014=1066.197,379.185,391.296,174.907,34.938,156.495
C08015=1066.190,378.939,391.335,174.903,34.931,156.493
C08016=1066.183,378.691,391.375,174.898,34.924,156.492
C08017=1066.175,378.445,391.414,174.894,34.918,156.490
C08018=1066.169,378.198,391.453,174.889,34.911,156.489
C08019=1066.162,377.952,391.492,174.884,34.904,156.487
C08020=1066.155,377.705,391.531,174.879,34.897,156.486
C08021=1066.147,377.458,391.571,174.874,34.891,156.484
C08022=1066.140,377.211,391.609,174.870,34.884,156.483
C08023=1066.133,376.965,391.649,174.865,34.877,156.481
C08024=1066.127,376.718,391.688,174.861,34.871,156.480
C08025=1066.120,376.471,391.727,174.856,34.864,156.478
C08026=1066.113,376.224,391.766,174.852,34.858,156.477
C08027=1066.105,375.977,391.805,174.847,34.851,156.475
C08028=1066.098,375.731,391.844,174.843,34.844,156.474
C08029=1066.092,375.484,391.883,174.838,34.837,156.472
C08030=1066.085,375.237,391.922,174.833,34.831,156.471
C08031=1066.078,374.990,391.961,174.828,34.824,156.470
C08032=1066.071,374.743,392.000,174.824,34.818,156.468
C08033=1066.064,374.496,392.039,174.819,34.812,156.467
C08034=1066.058,374.250,392.077,174.815,34.805,156.465
C08035=1066.050,374.003,392.116,174.810,34.799,156.464
C08036=1066.044,373.760,392.154,174.806,34.792,156.462
C08037=1066.036,373.517,392.192,174.801,34.786,156.461
C08038=1066.030,373.274,392.231,174.797,34.779,156.459
C08039=1066.023,373.031,392.268,174.792,34.773,156.458
C08040=1066.017,372.788,392.307,174.788,34.767,156.457
C08041=1066.009,372.544,392.345,174.784,34.760,156.455
C08042=1066.002,372.301,392.383,174.779,34.754,156.454
C08043=1065.995,372.058,392.420,174.775,34.748,156.452
C08044=1065.989,371.811,392.459,174.770,34.741,156.451
C08045=1065.982,371.564,392.498,174.766,34.735,156.450
C08046=1065.974,371.317,392.535,174.761,34.729,156.448
C08047=1065.968,371.070,392.574,174.757,34.723,156.447
C08048=1065.961,370.823,392.613,174.752,34.716,156.445
C08049=1065.954,370.576,392.651,174.748,34.710,156.444
C08050=1065.947,370.329,392.689,174.744,34.704,156.443
C08051=1065.940,370.084,392.727,174.739,34.698,156.441
C08052=1065.933,369.836,392.765,174.735,34.691,156.440
C08053=1065.927,369.589,392.804,174.730,34.685,156.439
C08054=1065.919,369.342,392.842,174.726,34.679,156.437
C08055=1065.912,369.095,392.881,174.721,34.672,156.436
C08056=1065.905,368.848,392.918,174.717,34.667,156.435
C08057=1065.898,368.601,392.957,174.713,34.660,156.433
C08058=1065.892,368.354,392.995,174.708,34.654,156.432
C08059=1065.885,368.107,393.033,174.705,34.648,156.430
C08060=1065.878,367.861,393.071,174.700,34.642,156.429
C08061=1065.871,367.614,393.109,174.696,34.636,156.428
C08062=1065.864,367.367,393.147,174.691,34.629,156.426
C08063=1065.858,367.119,393.186,174.687,34.623,156.425
C08064=1065.851,366.872,393.223,174.683,34.618,156.424
C08065=1065.845,366.625,393.261,174.678,34.611,156.422
C08066=1065.837,366.379,393.299,174.674,34.605,156.421
C08067=1065.831,366.131,393.337,174.669,34.599,156.420
C08068=1065.823,365.884,393.375,174.665,34.593,156.418
C08069=1065.818,365.638,393.412,174.661,34.587,156.417
C08070=1065.810,365.391,393.451,174.656,34.581,156.416
C08071=1065.803,365.144,393.489,174.653,34.575,156.414
C08072=1065.796,364.896,393.526,174.648,34.569,156.413
C08073=1065.790,364.650,393.564,174.644,34.563,156.412
C08074=1065.783,364.403,393.602,174.640,34.557,156.410
C08075=1065.777,364.155,393.640,174.635,34.551,156.409
C08076=1065.770,363.909,393.677,174.631,34.545,156.408
C08077=1065.763,363.662,393.714,174.627,34.539,156.406
C08078=1065.756,363.414,393.753,174.622,34.533,156.405
C08079=1065.750,363.168,393.790,174.619,34.527,156.404
C08080=1065.742,362.921,393.827,174.614,34.521,156.403
C08081=1065.736,362.673,393.865,174.610,34.515,156.401
C08082=1065.729,362.426,393.903,174.606,34.510,156.400
C08083=1065.722,362.179,393.939,174.601,34.503,156.399
C08084=1065.715,361.932,393.977,174.597,34.498,156.398
C08085=1065.709,361.685,394.015,174.594,34.492,156.396
C08086=1065.702,361.438,394.052,174.589,34.486,156.395
C08087=1065.695,361.191,394.090,174.585,34.480,156.394
C08088=1065.688,360.944,394.126,174.581,34.474,156.392
C08089=1065.682,360.696,394.164,174.576,34.469,156.391
C08090=1065.674,360.449,394.202,174.572,34.463,156.390
C08091=1065.668,360.202,394.238,174.569,34.457,156.389
C08092=1065.661,359.968,394.274,174.564,34.451,156.388
C08093=1065.656,359.734,394.310,174.560,34.446,156.386
C08094=1065.649,359.499,394.345,174.557,34.441,156.385
C08095=1065.643,359.265,394.380,174.552,34.435,156.384
C08096=1065.637,359.030,394.415,174.549,34.430,156.383
C08097=1065.630,358.795,394.450,174.545,34.424,156.382
C08098=1065.624,358.562,394.485,174.540,34.419,156.381
C08099=1065.617,358.327,394.520,174.537,34.413,156.379
C08100=1065.610,358.080,394.558,174.533,34.407,156.378
C08101=1065.603,357.833,394.594,174.528,34.402,156.377
C08102=1065.597,357.586,394.632,174.525,34.397,156.376
C08103=1065.590,357.338,394.668,174.521,34.391,156.374
C08104=1065.583,357.091,394.705,174.516,34.385,156.373
C08105=1065.576,356.844,394.742,174.512,34.379,156.372
C08106=1065.570,356.597,394.779,174.508,34.374,156.371
C08107=1065.563,356.349,394.816,174.504,34.368,156.370
C08108=1065.556,356.103,394.853,174.500,34.363,156.368
C08109=1065.549,355.855,394.890,174.496,34.357,156.367
C08110=1065.543,355.608,394.926,174.492,34.351,156.366
C08111=1065.536,355.362,394.963,174.488,34.346,156.365
C08112=1065.529,355.114,395.000,174.484,34.340,156.364
C08113=1065.523,354.867,395.036,174.480,34.335,156.362
C08114=1065.516,354.619,395.073,174.476,34.329,156.361
C08115=1065.510,354.372,395.110,174.472,34.324,156.360
C08116=1065.503,354.126,395.147,174.468,34.318,156.359
C08117=1065.496,353.878,395.184,174.464,34.313,156.358
C08118=1065.490,353.631,395.220,174.460,34.307,156.357
C08119=1065.483,353.384,395.257,174.456,34.301,156.355
C08120=1065.476,353.136,395.293,174.451,34.296,156.354
C08121=1065.470,352.889,395.330,174.448,34.290,156.353
C08122=1065.464,352.642,395.366,174.444,34.285,156.352
C08123=1065.457,352.394,395.403,174.440,34.279,156.351
C08124=1065.451,352.147,395.440,174.436,34.274,156.350
C08125=1065.444,351.900,395.476,174.432,34.269,156.348
C08126=1065.436,351.653,395.512,174.428,34.263,156.347
C08127=1065.430,351.406,395.549,174.424,34.258,156.346
C08128=1065.424,351.159,395.585,174.420,34.252,156.345
C08129=1065.417,350.911,395.622,174.416,34.247,156.344
C08130=1065.410,350.663,395.657,174.413,34.241,156.343
C08131=1065.404,350.416,395.693,174.408,34.236,156.342
C08132=1065.397,350.169,395.730,174.405,34.231,156.340
C08133=1065.391,349.922,395.767,174.401,34.225,156.339
C08134=1065.383,349.675,395.803,174.397,34.220,156.338
C08135=1065.377,349.427,395.838,174.393,34.215,156.337
C08136=1065.371,349.180,395.875,174.389,34.210,156.336
C08137=1065.363,348.933,395.911,174.385,34.204,156.335
C08138=1065.357,348.685,395.947,174.382,34.199,156.334
C08139=1065.351,348.438,395.983,174.377,34.194,156.333
C08140=1065.344,348.191,396.019,174.374,34.188,156.331
C08141=1065.338,347.944,396.055,174.370,34.183,156.330
C08142=1065.331,347.696,396.092,174.365,34.177,156.329
C08143=1065.324,347.449,396.127,174.362,34.172,156.328
C08144=1065.318,347.201,396.163,174.358,34.167,156.327
C08145=1065.312,346.954,396.200,174.355,34.162,156.326
C08146=1065.305,346.707,396.235,174.351,34.157,156.325
C08147=1065.298,346.460,396.271,174.346,34.151,156.324
C08148=1065.292,346.227,396.305,174.343,34.146,156.323
C08149=1065.286,345.995,396.338,174.340,34.141,156.322
C08150=1065.280,345.762,396.372,174.336,34.136,156.320
C08151=1065.274,345.530,396.405,174.332,34.132,156.319
C08152=1065.268,345.298,396.439,174.329,34.126,156.318
C08153=1065.261,345.065,396.473,174.325,34.122,156.317
C08154=1065.255,344.833,396.507,174.322,34.117,156.316
C08155=1065.249,344.600,396.541,174.318,34.112,156.315
C08156=1065.242,344.353,396.576,174.314,34.107,156.314
C08157=1065.236,344.105,396.611,174.311,34.102,156.313
C08158=1065.229,343.858,396.647,174.307,34.096,156.312
C08159=1065.223,343.611,396.683,174.303,34.091,156.311
C08160=1065.216,343.363,396.718,174.299,34.086,156.310
C08161=1065.210,343.116,396.755,174.295,34.081,156.309
C08162=1065.203,342.869,396.790,174.292,34.076,156.308
C08163=1065.197,342.622,396.825,174.288,34.071,156.307
C08164=1065.191,342.374,396.861,174.284,34.066,156.306
C08165=1065.184,342.127,396.896,174.280,34.061,156.305
C08166=1065.177,341.879,396.931,174.277,34.056,156.304
C08167=1065.171,341.632,396.967,174.273,34.050,156.302
C08168=1065.164,341.385,397.002,174.270,34.046,156.302
C08169=1065.157,341.137,397.038,174.265,34.040,156.300
C08170=1065.151,340.890,397.073,174.262,34.035,156.299
C08171=1065.144,340.642,397.108,174.258,34.031,156.298
C08172=1065.138,340.395,397.144,174.255,34.025,156.297
C08173=1065.132,340.147,397.179,174.250,34.020,156.296
C08174=1065.125,339.900,397.214,174.247,34.015,156.295
C08175=1065.118,339.653,397.250,174.243,34.010,156.294
C08176=1065.112,339.405,397.285,174.240,34.005,156.293
C08177=1065.105,339.157,397.320,174.236,34.000,156.292
C08178=1065.099,338.910,397.355,174.232,33.995,156.291
C08179=1065.093,338.663,397.390,174.228,33.990,156.290
C08180=1065.087,338.415,397.425,174.225,33.985,156.289
C08181=1065.080,338.168,397.461,174.222,33.980,156.288
C08182=1065.073,337.921,397.496,174.218,33.975,156.287
C08183=1065.067,337.673,397.531,174.214,33.970,156.286
C08184=1065.060,337.425,397.566,174.210,33.965,156.285
C08185=1065.054,337.177,397.601,174.207,33.960,156.284
C08186=1065.048,336.931,397.636,174.203,33.955,156.283
C08187=1065.041,336.683,397.671,174.200,33.950,156.282
C08188=1065.035,336.435,397.706,174.196,33.945,156.281
C08189=1065.028,336.188,397.741,174.192,33.941,156.280
C08190=1065.022,335.940,397.776,174.189,33.935,156.279
C08191=1065.015,335.692,397.811,174.185,33.931,156.278
C08192=1065.008,335.445,397.846,174.182,33.926,156.277
C08193=1065.002,335.198,397.880,174.178,33.921,156.276
C08194=1064.996,334.950,397.915,174.174,33.916,156.275
C08195=1064.989,334.703,397.950,174.170,33.911,156.274
C08196=1064.982,334.455,397.984,174.167,33.906,156.273
C08197=1064.976,334.208,398.020,174.164,33.902,156.272
C08198=1064.970,333.960,398.054,174.160,33.897,156.271
C08199=1064.963,333.713,398.089,174.157,33.892,156.270
C08200=1064.957,333.465,398.123,174.152,33.887,156.269
C08201=1064.950,333.218,398.158,174.149,33.882,156.268
C08202=1064.944,332.970,398.192,174.146,33.877,156.267
C08203=1064.937,332.723,398.227,174.142,33.872,156.266
C08204=1064.931,332.488,398.260,174.139,33.868,156.265
C08205=1064.926,332.254,398.293,174.136,33.863,156.264
C08206=1064.920,332.019,398.326,174.132,33.859,156.263
C08207=1064.913,331.784,398.359,174.129,33.854,156.262
C08208=1064.907,331.549,398.392,174.125,33.849,156.261
C08209=1064.901,331.315,398.424,174.122,33.845,156.260
C08210=1064.895,331.079,398.456,174.119,33.840,156.259
C08211=1064.890,330.844,398.490,174.116,33.836,156.258
C08212=1064.882,330.597,398.524,174.112,33.831,156.257
C08213=1064.876,330.350,398.558,174.108,33.826,156.256
C08214=1064.870,330.102,398.593,174.105,33.822,156.255
C08215=1064.863,329.854,398.626,174.101,33.817,156.254
C08216=1064.856,329.606,398.661,174.098,33.812,156.253
C08217=1064.850,329.359,398.695,174.095,33.808,156.253
C08218=1064.843,329.112,398.729,174.091,33.803,156.252
C08219=1064.836,328.864,398.764,174.087,33.799,156.251
C08220=1064.830,328.616,398.798,174.084,33.794,156.250
C08221=1064.823,328.369,398.832,174.080,33.789,156.249
C08222=1064.817,328.121,398.866,174.077,33.785,156.248
C08223=1064.811,327.873,398.900,174.074,33.780,156.247
C08224=1064.804,327.626,398.934,174.070,33.775,156.246
C08225=1064.797,327.378,398.968,174.066,33.770,156.245
C08226=1064.791,327.131,399.002,174.063,33.766,156.244
C08227=1064.784,326.883,399.036,174.059,33.762,156.243
C08228=1064.778,326.636,399.070,174.056,33.757,156.242
C08229=1064.771,326.388,399.104,174.053,33.752,156.241
C08230=1064.765,326.140,399.139,174.050,33.747,156.240
C08231=1064.758,325.893,399.172,174.046,33.743,156.239
C08232=1064.752,325.644,399.206,174.042,33.738,156.238
C08233=1064.746,325.397,399.240,174.039,33.734,156.238
C08234=1064.739,325.149,399.274,174.035,33.729,156.237
C08235=1064.733,324.902,399.308,174.032,33.724,156.236
C08236=1064.726,324.654,399.341,174.029,33.720,156.235
C08237=1064.720,324.407,399.376,174.026,33.716,156.234
C08238=1064.714,324.159,399.409,174.022,33.711,156.233
C08239=1064.707,323.912,399.443,174.019,33.706,156.232
C08240=1064.701,323.664,399.477,174.015,33.701,156.231
C08241=1064.694,323.417,399.511,174.012,33.697,156.230
C08242=1064.688,323.168,399.544,174.008,33.692,156.229
C08243=1064.681,322.921,399.578,174.005,33.688,156.228
C08244=1064.675,322.673,399.612,174.002,33.683,156.227
C08245=1064.668,322.426,399.646,173.999,33.679,156.227
C08246=1064.663,322.178,399.679,173.995,33.674,156.226
C08247=1064.656,321.930,399.713,173.992,33.669,156.225
C08248=1064.650,321.683,399.746,173.988,33.665,156.224
C08249=1064.644,321.435,399.781,173.985,33.661,156.223
C08250=1064.637,321.188,399.814,173.982,33.656,156.222
C08251=1064.631,320.940,399.847,173.978,33.651,156.221
C08252=1064.624,320.692,399.881,173.975,33.647,156.220
C08253=1064.619,320.444,399.914,173.972,33.642,156.219
C08254=1064.612,320.197,399.948,173.969,33.637,156.218
C08255=1064.606,319.949,399.982,173.965,33.633,156.217
C08256=1064.599,319.702,400.015,173.961,33.628,156.216
C08257=1064.594,319.454,400.048,173.958,33.624,156.215
C08258=1064.587,319.206,400.082,173.955,33.620,156.215
C08259=1064.581,318.958,400.116,173.952,33.615,156.214
C08260=1064.574,318.721,400.148,173.949,33.611,156.213
C08261=1064.568,318.483,400.180,173.946,33.606,156.212
C08262=1064.563,318.245,400.212,173.943,33.602,156.211
C08263=1064.556,318.008,400.244,173.940,33.598,156.210
C08264=1064.550,317.769,400.276,173.937,33.594,156.209
C08265=1064.545,317.532,400.308,173.932,33.589,156.208
C08266=1064.538,317.295,400.340,173.929,33.585,156.208
C08267=1064.533,317.057,400.372,173.926,33.580,156.207
C08268=1064.527,316.809,400.405,173.923,33.576,156.206
C08269=1064.520,316.561,400.439,173.920,33.571,156.205
C08270=1064.514,316.313,400.472,173.917,33.567,156.204
C08271=1064.508,316.066,400.505,173.914,33.562,156.203
C08272=1064.502,315.818,400.538,173.911,33.558,156.202
C08273=1064.496,315.571,400.572,173.908,33.553,156.201
C08274=1064.490,315.323,400.604,173.904,33.549,156.201
C08275=1064.484,315.075,400.638,173.900,33.544,156.200
C08276=1064.477,314.827,400.671,173.897,33.540,156.199
C08277=1064.471,314.580,400.704,173.894,33.535,156.198
C08278=1064.465,314.332,400.738,173.891,33.531,156.197
C08279=1064.459,314.085,400.770,173.888,33.526,156.196
C08280=1064.453,313.837,400.803,173.885,33.522,156.195
C08281=1064.446,313.589,400.836,173.882,33.518,156.194
C08282=1064.439,313.341,400.869,173.878,33.513,156.193
C08283=1064.433,313.094,400.902,173.875,33.509,156.193
C08284=1064.427,312.846,400.935,173.872,33.505,156.192
C08285=1064.420,312.598,400.967,173.869,33.500,156.191
C08286=1064.414,312.350,401.000,173.865,33.496,156.190
C08287=1064.407,312.102,401.033,173.862,33.492,156.189
C08288=1064.401,311.855,401.066,173.859,33.488,156.188
C08289=1064.395,311.607,401.099,173.856,33.483,156.188
C08290=1064.389,311.359,401.131,173.852,33.479,156.187
C08291=1064.382,311.111,401.164,173.849,33.474,156.186
C08292=1064.376,310.863,401.196,173.846,33.470,156.185
C08293=1064.369,310.616,401.229,173.843,33.466,156.184
C08294=1064.362,310.368,401.261,173.840,33.462,156.183
C08295=1064.356,310.121,401.294,173.837,33.457,156.182
C08296=1064.350,309.873,401.326,173.834,33.453,156.182
C08297=1064.344,309.625,401.359,173.831,33.449,156.181
C08298=1064.337,309.377,401.392,173.827,33.445,156.180
C08299=1064.331,309.130,401.424,173.823,33.440,156.179
C08300=1064.325,308.882,401.457,173.820,33.436,156.178
C08301=1064.318,308.633,401.489,173.817,33.431,156.177
C08302=1064.312,308.386,401.522,173.814,33.427,156.176
C08303=1064.305,308.138,401.554,173.811,33.423,156.176
C08304=1064.299,307.890,401.586,173.808,33.419,156.175
C08305=1064.293,307.643,401.619,173.805,33.415,156.174
C08306=1064.286,307.395,401.652,173.802,33.410,156.173
C08307=1064.280,307.147,401.684,173.799,33.406,156.172
C08308=1064.274,306.899,401.717,173.796,33.401,156.171
C08309=1064.267,306.652,401.749,173.793,33.397,156.171
C08310=1064.261,306.404,401.781,173.790,33.393,156.170
C08311=1064.255,306.156,401.814,173.787,33.389,156.169
C08312=1064.249,305.908,401.846,173.783,33.385,156.168
C08313=1064.243,305.661,401.878,173.780,33.381,156.167
C08314=1064.237,305.413,401.910,173.777,33.376,156.167
C08315=1064.230,305.165,401.942,173.773,33.372,156.166
C08316=1064.224,304.929,401.974,173.771,33.368,156.165
C08317=1064.218,304.693,402.004,173.768,33.364,156.164
C08318=1064.212,304.458,402.034,173.765,33.360,156.163
C08319=1064.207,304.222,402.065,173.762,33.356,156.163
C08320=1064.200,303.986,402.096,173.759,33.352,156.162
C08321=1064.195,303.750,402.126,173.756,33.347,156.161
C08322=1064.189,303.514,402.157,173.753,33.343,156.160
C08323=1064.182,303.278,402.188,173.750,33.340,156.159
C08324=1064.177,303.030,402.220,173.747,33.335,156.159
C08325=1064.171,302.783,402.252,173.744,33.331,156.158
C08326=1064.164,302.535,402.284,173.741,33.326,156.157
C08327=1064.158,302.287,402.316,173.738,33.322,156.156
C08328=1064.152,302.039,402.348,173.734,33.318,156.155
C08329=1064.146,301.791,402.380,173.732,33.314,156.154
C08330=1064.140,301.544,402.412,173.729,33.310,156.153
C08331=1064.133,301.296,402.444,173.726,33.306,156.153
C08332=1064.127,301.048,402.476,173.723,33.301,156.152
C08333=1064.121,300.800,402.508,173.720,33.297,156.151
C08334=1064.115,300.552,402.540,173.717,33.293,156.150
C08335=1064.109,300.305,402.572,173.714,33.289,156.149
C08336=1064.103,300.057,402.604,173.711,33.284,156.149
C08337=1064.097,299.808,402.636,173.708,33.280,156.148
C08338=1064.090,299.561,402.668,173.705,33.276,156.147
C08339=1064.085,299.313,402.699,173.702,33.272,156.146
C08340=1064.079,299.065,402.731,173.699,33.268,156.145
C08341=1064.073,298.817,402.764,173.696,33.263,156.144
C08342=1064.066,298.570,402.795,173.693,33.259,156.144
C08343=1064.060,298.322,402.827,173.690,33.254,156.143
C08344=1064.055,298.074,402.859,173.687,33.250,156.142
C08345=1064.048,297.826,402.891,173.684,33.246,156.141
C08346=1064.042,297.578,402.922,173.681,33.242,156.140
C08347=1064.036,297.330,402.954,173.678,33.238,156.139
C08348=1064.030,297.082,402.986,173.674,33.233,156.139
C08349=1064.024,296.835,403.017,173.672,33.229,156.138
C08350=1064.018,296.587,403.049,173.669,33.226,156.137
C08351=1064.012,296.338,403.081,173.666,33.221,156.136
C08352=1064.005,296.091,403.112,173.663,33.217,156.136
C08353=1063.999,295.843,403.144,173.660,33.213,156.135
C08354=1063.993,295.595,403.175,173.657,33.209,156.134
C08355=1063.987,295.347,403.207,173.654,33.204,156.133
C08356=1063.981,295.099,403.238,173.651,33.200,156.132
C08357=1063.974,294.851,403.269,173.648,33.197,156.132
C08358=1063.968,294.603,403.301,173.645,33.192,156.131
C08359=1063.962,294.356,403.332,173.642,33.188,156.130
C08360=1063.955,294.108,403.364,173.639,33.184,156.129
C08361=1063.950,293.859,403.395,173.637,33.180,156.128
C08362=1063.944,293.612,403.426,173.634,33.176,156.128
C08363=1063.937,293.364,403.458,173.631,33.172,156.127
C08364=1063.931,293.116,403.490,173.628,33.168,156.126
C08365=1063.925,292.868,403.520,173.625,33.163,156.125
C08366=1063.918,292.620,403.551,173.622,33.159,156.124
C08367=1063.912,292.372,403.583,173.619,33.155,156.124
C08368=1063.907,292.124,403.614,173.616,33.151,156.123
C08369=1063.900,291.876,403.645,173.613,33.147,156.122
C08370=1063.893,291.628,403.677,173.611,33.143,156.121
C08371=1063.888,291.380,403.708,173.608,33.139,156.120
C08372=1063.882,291.151,403.736,173.605,33.135,156.120
C08373=1063.877,290.923,403.765,173.602,33.131,156.119
C08374=1063.871,290.695,403.794,173.600,33.128,156.118
C08375=1063.865,290.467,403.822,173.597,33.124,156.118
C08376=1063.859,290.239,403.850,173.594,33.120,156.117
C08377=1063.853,290.010,403.879,173.592,33.116,156.116
C08378=1063.848,289.782,403.908,173.589,33.113,156.115
C08379=1063.842,289.554,403.936,173.586,33.109,156.115
C08380=1063.836,289.306,403.968,173.583,33.105,156.114
C08381=1063.830,289.058,403.998,173.580,33.101,156.113
C08382=1063.824,288.810,404.030,173.577,33.097,156.112
C08383=1063.817,288.562,404.061,173.574,33.093,156.112
C08384=1063.812,288.314,404.091,173.571,33.088,156.111
C08385=1063.805,288.066,404.123,173.568,33.085,156.110
C08386=1063.799,287.818,404.153,173.566,33.081,156.109
C08387=1063.792,287.570,404.185,173.563,33.076,156.108
C08388=1063.786,287.322,404.215,173.560,33.073,156.108
C08389=1063.780,287.074,404.246,173.557,33.068,156.107
C08390=1063.774,286.827,404.277,173.554,33.064,156.106
C08391=1063.768,286.578,404.307,173.551,33.060,156.105
C08392=1063.762,286.330,404.338,173.549,33.056,156.105
C08393=1063.755,286.082,404.369,173.546,33.053,156.104
C08394=1063.749,285.834,404.400,173.543,33.048,156.103
C08395=1063.743,285.586,404.430,173.540,33.044,156.102
C08396=1063.737,285.338,404.461,173.537,33.040,156.102
C08397=1063.730,285.090,404.492,173.535,33.036,156.101
C08398=1063.724,284.842,404.522,173.532,33.032,156.100
C08399=1063.718,284.594,404.553,173.529,33.028,156.099
C08400=1063.712,284.346,404.583,173.526,33.024,156.098
C08401=1063.706,284.098,404.614,173.523,33.020,156.098
C08402=1063.700,283.850,404.645,173.521,33.016,156.097
C08403=1063.693,283.602,404.676,173.518,33.012,156.096
C08404=1063.687,283.354,404.706,173.515,33.008,156.095
C08405=1063.682,283.106,404.737,173.512,33.004,156.095
C08406=1063.675,282.858,404.767,173.509,33.000,156.094
C08407=1063.669,282.610,404.798,173.507,32.996,156.093
C08408=1063.663,282.361,404.828,173.504,32.992,156.092
C08409=1063.657,282.113,404.859,173.501,32.988,156.092
C08410=1063.651,281.866,404.889,173.498,32.984,156.091
C08411=1063.645,281.617,404.920,173.496,32.980,156.090
C08412=1063.639,281.369,404.950,173.493,32.976,156.089
C08413=1063.632,281.121,404.980,173.490,32.972,156.089
C08414=1063.626,280.873,405.011,173.487,32.968,156.088
C08415=1063.620,280.625,405.041,173.485,32.964,156.087
C08416=1063.614,280.377,405.072,173.482,32.960,156.086
C08417=1063.608,280.129,405.102,173.479,32.955,156.085
C08418=1063.602,279.881,405.132,173.476,32.952,156.085
C08419=1063.596,279.633,405.163,173.474,32.948,156.084
C08420=1063.589,279.385,405.193,173.471,32.944,156.083
C08421=1063.583,279.137,405.223,173.468,32.940,156.082
C08422=1063.577,278.889,405.254,173.465,32.936,156.082
C08423=1063.571,278.641,405.284,173.463,32.932,156.081
C08424=1063.565,278.393,405.313,173.460,32.928,156.080
C08425=1063.559,278.144,405.344,173.457,32.924,156.079
C08426=1063.553,277.897,405.374,173.454,32.920,156.079
C08427=1063.546,277.649,405.404,173.452,32.916,156.078
C08428=1063.541,277.426,405.432,173.449,32.912,156.077
C08429=1063.535,277.203,405.458,173.447,32.909,156.077
C08430=1063.530,276.980,405.486,173.444,32.905,156.076
C08431=1063.524,276.757,405.512,173.442,32.902,156.075
C08432=1063.519,276.533,405.540,173.439,32.898,156.075
C08433=1063.513,276.310,405.566,173.437,32.895,156.074
C08434=1063.508,276.087,405.594,173.435,32.891,156.073
C08435=1063.502,275.864,405.620,173.432,32.887,156.073
C08436=1063.497,275.616,405.651,173.429,32.884,156.072
C08437=1063.490,275.368,405.681,173.427,32.879,156.071
C08438=1063.484,275.120,405.711,173.424,32.876,156.070
C08439=1063.477,274.872,405.740,173.421,32.871,156.070
C08440=1063.472,274.624,405.771,173.419,32.868,156.069
C08441=1063.466,274.376,405.800,173.416,32.864,156.068
C08442=1063.459,274.128,405.830,173.413,32.860,156.067
C08443=1063.453,273.879,405.860,173.411,32.856,156.067
C08444=1063.447,273.632,405.890,173.408,32.852,156.066
C08445=1063.441,273.383,405.919,173.405,32.848,156.065
C08446=1063.435,273.135,405.950,173.403,32.844,156.064
C08447=1063.428,272.887,405.980,173.400,32.840,156.064
C08448=1063.423,272.639,406.010,173.397,32.836,156.063
C08449=1063.417,272.391,406.039,173.395,32.832,156.062
C08450=1063.411,272.143,406.069,173.392,32.828,156.061
C08451=1063.404,271.894,406.098,173.389,32.824,156.061
C08452=1063.398,271.646,406.129,173.387,32.820,156.060
C08453=1063.392,271.398,406.158,173.384,32.816,156.059
C08454=1063.386,271.150,406.188,173.381,32.812,156.058
C08455=1063.380,270.902,406.217,173.379,32.808,156.058
C08456=1063.374,270.653,406.247,173.377,32.804,156.057
C08457=1063.367,270.405,406.277,173.374,32.800,156.056
C08458=1063.361,270.157,406.306,173.372,32.796,156.055
C08459=1063.355,269.909,406.336,173.369,32.793,156.055
C08460=1063.349,269.661,406.365,173.366,32.788,156.054
C08461=1063.343,269.413,406.395,173.364,32.785,156.053
C08462=1063.337,269.165,406.424,173.361,32.781,156.052
C08463=1063.331,268.917,406.454,173.358,32.777,156.052
C08464=1063.324,268.668,406.484,173.356,32.773,156.051
C08465=1063.318,268.420,406.513,173.353,32.769,156.050
C08466=1063.313,268.171,406.542,173.350,32.765,156.050
C08467=1063.306,267.923,406.571,173.348,32.761,156.049
C08468=1063.300,267.676,406.601,173.345,32.757,156.048
C08469=1063.294,267.428,406.630,173.343,32.753,156.047
C08470=1063.288,267.179,406.660,173.340,32.749,156.047
C08471=1063.282,266.931,406.689,173.337,32.745,156.046
C08472=1063.275,266.682,406.718,173.335,32.741,156.045
C08473=1063.269,266.434,406.748,173.332,32.738,156.044
C08474=1063.263,266.186,406.777,173.329,32.733,156.044
C08475=1063.257,265.938,406.807,173.327,32.730,156.043
C08476=1063.251,265.690,406.836,173.324,32.726,156.042
C08477=1063.245,265.442,406.865,173.322,32.722,156.041
C08478=1063.239,265.193,406.895,173.319,32.718,156.041
C08479=1063.232,264.945,406.924,173.316,32.714,156.040
C08480=1063.227,264.697,406.953,173.314,32.710,156.039
C08481=1063.221,264.449,406.982,173.311,32.706,156.038
C08482=1063.214,264.201,407.011,173.309,32.702,156.038
C08483=1063.208,263.952,407.040,173.306,32.698,156.037
C08484=1063.204,263.731,407.066,173.304,32.695,156.036
C08485=1063.198,263.510,407.092,173.301,32.691,156.036
C08486=1063.192,263.288,407.118,173.299,32.688,156.035
C08487=1063.186,263.068,407.144,173.297,32.685,156.034
C08488=1063.181,262.847,407.170,173.295,32.681,156.034
C08489=1063.175,262.626,407.196,173.293,32.677,156.033
C08490=1063.169,262.404,407.222,173.291,32.674,156.033
C08491=1063.164,262.183,407.247,173.289,32.670,156.032
C08492=1063.158,261.935,407.276,173.286,32.667,156.031
C08493=1063.151,261.686,407.305,173.283,32.663,156.030
C08494=1063.145,261.438,407.334,173.281,32.659,156.030
C08495=1063.139,261.190,407.363,173.278,32.655,156.029
C08496=1063.133,260.941,407.392,173.276,32.651,156.028
C08497=1063.127,260.693,407.421,173.273,32.648,156.028
C08498=1063.120,260.445,407.450,173.271,32.644,156.027
C08499=1063.114,260.197,407.479,173.268,32.640,156.026
C08500=1063.108,259.948,407.507,173.265,32.636,156.025
C08501=1063.102,259.700,407.536,173.263,32.632,156.025
C08502=1063.096,259.452,407.565,173.260,32.628,156.024
C08503=1063.089,259.204,407.594,173.258,32.624,156.023
C08504=1063.083,258.955,407.622,173.255,32.620,156.022
C08505=1063.077,258.707,407.651,173.253,32.616,156.022
C08506=1063.070,258.459,407.680,173.250,32.613,156.021
C08507=1063.064,258.210,407.708,173.248,32.609,156.020
C08508=1063.058,257.962,407.737,173.245,32.605,156.020
C08509=1063.052,257.714,407.766,173.242,32.601,156.019
C08510=1063.046,257.465,407.795,173.240,32.597,156.018
C08511=1063.040,257.217,407.824,173.237,32.593,156.017
C08512=1063.034,256.969,407.852,173.236,32.589,156.017
C08513=1063.027,256.721,407.880,173.233,32.586,156.016
C08514=1063.021,256.473,407.908,173.231,32.581,156.015
C08515=1063.015,256.225,407.937,173.228,32.578,156.015
C08516=1063.009,255.976,407.966,173.226,32.574,156.014
C08517=1063.003,255.728,407.995,173.223,32.570,156.013
C08518=1062.997,255.479,408.023,173.221,32.566,156.012
C08519=1062.991,255.231,408.052,173.218,32.562,156.012
C08520=1062.985,254.983,408.080,173.216,32.558,156.011
C08521=1062.978,254.735,408.109,173.213,32.554,156.010
C08522=1062.972,254.486,408.137,173.211,32.550,156.009
C08523=1062.966,254.238,408.166,173.208,32.546,156.009
C08524=1062.960,253.989,408.194,173.206,32.543,156.008
C08525=1062.954,253.741,408.223,173.203,32.538,156.007
C08526=1062.949,253.493,408.251,173.201,32.535,156.007
C08527=1062.942,253.245,408.280,173.198,32.531,156.006
C08528=1062.936,252.996,408.308,173.196,32.527,156.005
C08529=1062.930,252.748,408.336,173.193,32.523,156.005
C08530=1062.924,252.500,408.365,173.192,32.519,156.004
C08531=1062.918,252.252,408.393,173.189,32.515,156.003
C08532=1062.912,252.003,408.421,173.187,32.512,156.002
C08533=1062.905,251.755,408.450,173.184,32.507,156.002
C08534=1062.899,251.506,408.478,173.182,32.504,156.001
C08535=1062.894,251.258,408.506,173.180,32.499,156.000
C08536=1062.888,251.010,408.535,173.177,32.496,155.999
C08537=1062.882,250.761,408.564,173.175,32.491,155.999
C08538=1062.875,250.513,408.592,173.172,32.488,155.998
C08539=1062.870,250.265,408.619,173.170,32.484,155.997
C08540=1062.864,250.043,408.645,173.168,32.480,155.997
C08541=1062.859,249.820,408.671,173.165,32.477,155.996
C08542=1062.854,249.598,408.696,173.163,32.473,155.995
C08543=1062.848,249.376,408.721,173.161,32.470,155.995
C08544=1062.842,249.154,408.746,173.159,32.466,155.994
C08545=1062.838,248.931,408.772,173.157,32.462,155.993
C08546=1062.832,248.709,408.797,173.155,32.459,155.993
C08547=1062.827,248.486,408.822,173.153,32.456,155.992
C08548=1062.821,248.238,408.850,173.151,32.451,155.991
C08549=1062.815,247.990,408.879,173.148,32.448,155.991
C08550=1062.808,247.742,408.907,173.146,32.443,155.990
C08551=1062.803,247.494,408.934,173.144,32.440,155.989
C08552=1062.797,247.245,408.963,173.141,32.435,155.988
C08553=1062.792,246.997,408.991,173.139,32.432,155.988
C08554=1062.785,246.748,409.019,173.136,32.427,155.987
C08555=1062.779,246.500,409.047,173.134,32.424,155.986
C08556=1062.774,246.252,409.075,173.131,32.419,155.985
C08557=1062.767,246.003,409.103,173.129,32.416,155.985
C08558=1062.761,245.754,409.131,173.127,32.412,155.984
C08559=1062.755,245.507,409.158,173.124,32.408,155.983
C08560=1062.749,245.258,409.187,173.122,32.404,155.982
C08561=1062.742,245.009,409.214,173.120,32.400,155.982
C08562=1062.737,244.761,409.242,173.118,32.396,155.981
C08563=1062.731,244.513,409.271,173.116,32.392,155.980
C08564=1062.724,244.264,409.298,173.113,32.388,155.979
C08565=1062.719,244.016,409.326,173.111,32.384,155.979
C08566=1062.712,243.768,409.354,173.108,32.381,155.978
C08567=1062.707,243.519,409.381,173.106,32.376,155.977
C08568=1062.701,243.271,409.409,173.104,32.373,155.977
C08569=1062.695,243.022,409.437,173.101,32.368,155.976
C08570=1062.689,242.774,409.465,173.099,32.365,155.975
C08571=1062.683,242.525,409.493,173.096,32.361,155.975
C08572=1062.677,242.278,409.520,173.094,32.357,155.974
C08573=1062.670,242.028,409.547,173.092,32.353,155.973
C08574=1062.664,241.780,409.576,173.090,32.349,155.972
C08575=1062.658,241.532,409.603,173.088,32.345,155.972
C08576=1062.652,241.284,409.631,173.086,32.341,155.971
C08577=1062.647,241.035,409.658,173.083,32.337,155.970
C08578=1062.640,240.786,409.686,173.081,32.333,155.969
C08579=1062.633,240.538,409.713,173.078,32.330,155.969
C08580=1062.628,240.289,409.741,173.076,32.325,155.968
C08581=1062.621,240.041,409.768,173.074,32.322,155.967
C08582=1062.615,239.793,409.796,173.071,32.318,155.967
C08583=1062.610,239.544,409.823,173.069,32.314,155.966
C08584=1062.604,239.296,409.851,173.067,32.310,155.965
C08585=1062.597,239.048,409.878,173.065,32.306,155.964
C08586=1062.591,238.799,409.905,173.063,32.302,155.964
C08587=1062.585,238.550,409.933,173.061,32.298,155.963
C08588=1062.579,238.302,409.961,173.058,32.295,155.962
C08589=1062.573,238.054,409.988,173.056,32.290,155.961
C08590=1062.566,237.805,410.016,173.053,32.287,155.961
C08591=1062.560,237.557,410.042,173.051,32.283,155.960
C08592=1062.554,237.308,410.071,173.049,32.279,155.959
C08593=1062.549,237.060,410.097,173.046,32.275,155.959
C08594=1062.542,236.811,410.125,173.044,32.271,155.958
C08595=1062.536,236.563,410.152,173.042,32.267,155.957
C08596=1062.531,236.337,410.177,173.040,32.263,155.957
C08597=1062.525,236.112,410.201,173.039,32.260,155.956
C08598=1062.520,235.887,410.226,173.036,32.256,155.955
C08599=1062.514,235.662,410.250,173.034,32.253,155.955
C08600=1062.509,235.436,410.275,173.032,32.249,155.954
C08601=1062.503,235.211,410.300,173.030,32.245,155.953
C08602=1062.498,234.986,410.325,173.028,32.242,155.953
C08603=1062.493,234.760,410.350,173.026,32.239,155.952
C08604=1062.486,234.511,410.377,173.024,32.234,155.951
C08605=1062.480,234.263,410.404,173.021,32.231,155.951
C08606=1062.474,234.014,410.431,173.019,32.226,155.950
C08607=1062.468,233.766,410.459,173.017,32.223,155.949
C08608=1062.463,233.518,410.486,173.015,32.218,155.948
C08609=1062.456,233.269,410.513,173.013,32.215,155.948
C08610=1062.450,233.021,410.540,173.011,32.211,155.947
C08611=1062.444,232.772,410.567,173.008,32.207,155.946
C08612=1062.438,232.524,410.594,173.006,32.203,155.945
C08613=1062.432,232.276,410.621,173.004,32.199,155.945
C08614=1062.426,232.027,410.648,173.002,32.195,155.944
C08615=1062.420,231.778,410.675,172.999,32.191,155.943
C08616=1062.413,231.529,410.702,172.997,32.187,155.942
C08617=1062.407,231.282,410.729,172.996,32.183,155.942
C08618=1062.402,231.033,410.756,172.993,32.179,155.941
C08619=1062.395,230.784,410.783,172.991,32.175,155.940
C08620=1062.389,230.536,410.810,172.989,32.171,155.940
C08621=1062.384,230.288,410.836,172.987,32.167,155.939
C08622=1062.377,230.039,410.864,172.984,32.163,155.938
C08623=1062.371,229.791,410.891,172.982,32.159,155.937
C08624=1062.365,229.542,410.917,172.980,32.155,155.937
C08625=1062.359,229.293,410.944,172.978,32.151,155.936
C08626=1062.353,229.045,410.971,172.975,32.147,155.935
C08627=1062.347,228.796,410.998,172.974,32.144,155.935
C08628=1062.341,228.565,411.023,172.972,32.140,155.934
C08629=1062.335,228.334,411.048,172.970,32.136,155.933
C08630=1062.330,228.101,411.073,172.968,32.133,155.933
C08631=1062.325,227.870,411.097,172.966,32.129,155.932
C08632=1062.318,227.639,411.122,172.963,32.125,155.931
C08633=1062.312,227.407,411.147,172.961,32.122,155.931
C08634=1062.307,227.175,411.172,172.959,32.118,155.930
C08635=1062.301,226.944,411.196,172.957,32.114,155.929
C08636=1062.295,226.695,411.223,172.956,32.110,155.929
C08637=1062.289,226.447,411.250,172.954,32.106,155.928
C08638=1062.283,226.198,411.277,172.951,32.102,155.927
C08639=1062.277,225.949,411.304,172.949,32.099,155.926
C08640=1062.271,225.701,411.330,172.947,32.094,155.926
C08641=1062.265,225.453,411.356,172.945,32.091,155.925
C08642=1062.259,225.205,411.383,172.942,32.086,155.924
C08643=1062.253,224.955,411.410,172.940,32.083,155.923
C08644=1062.246,224.707,411.436,172.938,32.078,155.923
C08645=1062.240,224.459,411.463,172.937,32.075,155.922
C08646=1062.235,224.211,411.489,172.935,32.070,155.921
C08647=1062.228,223.962,411.516,172.932,32.067,155.921
C08648=1062.222,223.713,411.543,172.930,32.063,155.920
C08649=1062.216,223.465,411.568,172.928,32.059,155.919
C08650=1062.210,223.216,411.595,172.926,32.055,155.918
C08651=1062.204,222.967,411.622,172.923,32.051,155.918
C08652=1062.198,222.721,411.648,172.921,32.047,155.917
C08653=1062.192,222.474,411.674,172.920,32.043,155.916
C08654=1062.187,222.228,411.701,172.918,32.039,155.915
C08655=1062.180,221.982,411.727,172.916,32.035,155.915
C08656=1062.175,221.736,411.753,172.914,32.031,155.914
C08657=1062.169,221.489,411.779,172.911,32.027,155.913
C08658=1062.163,221.243,411.805,172.909,32.023,155.913
C08659=1062.156,220.997,411.831,172.907,32.019,155.912
C08660=1062.150,220.748,411.858,172.905,32.015,155.911
C08661=1062.144,220.500,411.883,172.903,32.011,155.910
C08662=1062.138,220.251,411.910,172.901,32.007,155.910
C08663=1062.132,220.003,411.936,172.899,32.003,155.909
C08664=1062.126,219.754,411.962,172.897,31.999,155.908
C08665=1062.120,219.505,411.989,172.895,31.995,155.907
C08666=1062.113,219.257,412.015,172.893,31.992,155.907
C08667=1062.108,219.008,412.041,172.890,31.987,155.906
C08668=1062.101,218.760,412.067,172.888,31.983,155.905
C08669=1062.095,218.511,412.094,172.887,31.979,155.905
C08670=1062.089,218.262,412.119,172.885,31.975,155.904
C08671=1062.083,218.014,412.146,172.883,31.971,155.903
C08672=1062.077,217.765,412.171,172.881,31.967,155.902
C08673=1062.071,217.517,412.198,172.878,31.963,155.902
C08674=1062.065,217.268,412.223,172.876,31.959,155.901
C08675=1062.059,217.020,412.250,172.874,31.955,155.900
C08676=1062.052,216.771,412.276,172.872,31.951,155.899
C08677=1062.046,216.522,412.302,172.871,31.947,155.899
C08678=1062.040,216.274,412.328,172.869,31.943,155.898
C08679=1062.034,216.025,412.354,172.866,31.939,155.897
C08680=1062.028,215.777,412.380,172.864,31.935,155.897
C08681=1062.022,215.529,412.406,172.862,31.931,155.896
C08682=1062.016,215.280,412.432,172.860,31.927,155.895
C08683=1062.010,215.031,412.458,172.858,31.923,155.894
C08684=1062.004,214.783,412.484,172.857,31.919,155.894
C08685=1061.998,214.534,412.510,172.855,31.915,155.893
C08686=1061.992,214.285,412.535,172.852,31.911,155.892
C08687=1061.986,214.037,412.562,172.850,31.907,155.891
C08688=1061.980,213.788,412.587,172.848,31.903,155.891
C08689=1061.974,213.540,412.613,172.846,31.899,155.890
C08690=1061.968,213.291,412.639,172.844,31.895,155.889
C08691=1061.962,213.043,412.665,172.843,31.891,155.888
C08692=1061.956,212.794,412.690,172.841,31.887,155.888
C08693=1061.950,212.545,412.717,172.839,31.883,155.887
C08694=1061.943,212.296,412.742,172.836,31.879,155.886
C08695=1061.937,212.048,412.768,172.834,31.875,155.886
C08696=1061.931,211.799,412.794,172.832,31.871,155.885
C08697=1061.925,211.551,412.820,172.830,31.867,155.884
C08698=1061.919,211.302,412.845,172.829,31.863,155.883
C08699=1061.914,211.053,412.871,172.827,31.858,155.882
C08700=1061.907,210.805,412.897,172.825,31.855,155.882
C08701=1061.901,210.556,412.922,172.823,31.850,155.881
C08702=1061.895,210.307,412.948,172.820,31.846,155.880
C08703=1061.889,210.059,412.974,172.818,31.842,155.880
C08704=1061.883,209.811,413.000,172.816,31.838,155.879
C08705=1061.876,209.562,413.025,172.815,31.834,155.878
C08706=1061.870,209.313,413.050,172.813,31.830,155.877
C08707=1061.865,209.064,413.076,172.811,31.826,155.877
C08708=1061.859,208.838,413.099,172.809,31.822,155.876
C08709=1061.853,208.611,413.122,172.807,31.819,155.875
C08710=1061.848,208.384,413.146,172.805,31.815,155.875
C08711=1061.842,208.157,413.169,172.803,31.811,155.874
C08712=1061.837,207.930,413.193,172.802,31.808,155.873
C08713=1061.831,207.703,413.216,172.801,31.804,155.873
C08714=1061.826,207.477,413.239,172.799,31.800,155.872
C08715=1061.820,207.249,413.263,172.797,31.797,155.871
C08716=1061.795,206.201,413.366,172.623,31.714,155.863
C08717=1061.790,205.952,413.390,172.621,31.711,155.863
C08718=1061.784,205.704,413.416,172.619,31.707,155.862
C08719=1061.778,205.455,413.440,172.616,31.704,155.862
C08720=1061.772,205.206,413.465,172.614,31.701,155.861
C08721=1061.766,204.958,413.489,172.611,31.698,155.860
C08722=1061.760,204.709,413.514,172.610,31.694,155.860
C08723=1061.755,204.460,413.538,172.607,31.691,155.859
C08724=1061.749,204.212,413.563,172.605,31.688,155.859
C08725=1061.743,203.962,413.588,172.603,31.685,155.858
C08726=1061.737,203.714,413.612,172.600,31.682,155.858
C08727=1061.731,203.465,413.636,172.598,31.678,155.857
C08728=1061.725,203.217,413.661,172.595,31.676,155.857
C08729=1061.720,202.968,413.685,172.594,31.672,155.856
C08730=1061.714,202.719,413.710,172.592,31.669,155.856
C08731=1061.709,202.470,413.734,172.589,31.666,155.855
C08732=1061.703,202.221,413.759,172.587,31.663,155.855
C08733=1061.696,201.973,413.783,172.585,31.660,155.854
C08734=1061.691,201.724,413.808,172.582,31.656,155.854
C08735=1061.685,201.476,413.832,172.581,31.654,155.853
C08736=1061.679,201.226,413.856,172.578,31.650,155.853
C08737=1061.673,200.978,413.880,172.576,31.647,155.852
C08738=1061.667,200.729,413.904,172.574,31.644,155.852
C08739=1061.661,200.480,413.929,172.571,31.641,155.851
C08740=1061.655,200.231,413.953,172.569,31.638,155.851
C08741=1061.649,199.983,413.977,172.566,31.635,155.850
C08742=1061.643,199.734,414.001,172.565,31.632,155.850
C08743=1061.638,199.485,414.025,172.563,31.629,155.849
C08744=1061.631,199.237,414.050,172.560,31.626,155.849
C08745=1061.625,198.988,414.074,172.558,31.623,155.848
C08746=1061.619,198.739,414.098,172.556,31.620,155.848
C08747=1061.613,198.491,414.123,172.553,31.617,155.847
C08748=1061.607,198.241,414.146,172.551,31.614,155.847
C08749=1061.602,197.992,414.170,172.549,31.610,155.846
C08750=1061.595,197.743,414.194,172.547,31.608,155.846
C08751=1061.590,197.495,414.218,172.545,31.604,155.845
C08752=1061.584,197.247,414.242,172.542,31.601,155.845
C08753=1061.578,196.997,414.267,172.540,31.599,155.844
C08754=1061.572,196.749,414.290,172.538,31.595,155.844
C08755=1061.566,196.500,414.315,172.536,31.592,155.843
C08756=1061.560,196.252,414.339,172.534,31.589,155.843
C08757=1061.555,196.003,414.363,172.532,31.586,155.842
C08758=1061.548,195.754,414.387,172.529,31.583,155.842
C08759=1061.543,195.505,414.411,172.527,31.580,155.841
C08760=1061.536,195.256,414.435,172.525,31.577,155.841
C08761=1061.531,195.007,414.459,172.522,31.574,155.840
C08762=1061.525,194.759,414.482,172.521,31.571,155.839
C08763=1061.519,194.510,414.507,172.519,31.568,155.839
C08764=1061.513,194.261,414.531,172.516,31.565,155.839
C08765=1061.508,194.013,414.555,172.514,31.562,155.838
C08766=1061.501,193.763,414.578,172.512,31.559,155.838
C08767=1061.496,193.515,414.603,172.509,31.556,155.837
C08768=1061.490,193.266,414.626,172.508,31.552,155.836
C08769=1061.484,193.017,414.651,172.506,31.550,155.836
C08770=1061.478,192.768,414.674,172.503,31.547,155.836
C08771=1061.472,192.520,414.697,172.501,31.543,155.835
C08772=1061.466,192.271,414.722,172.499,31.541,155.835
C08773=1061.460,192.022,414.746,172.497,31.538,155.834
C08774=1061.455,191.773,414.769,172.494,31.534,155.833
C08775=1061.449,191.525,414.793,172.493,31.532,155.833
C08776=1061.444,191.275,414.818,172.491,31.528,155.833
C08777=1061.437,190.992,414.844,172.488,31.525,155.832
C08778=1061.430,190.709,414.871,172.485,31.521,155.831
C08779=1061.424,190.425,414.898,172.483,31.518,155.831
C08780=1061.418,190.142,414.926,172.481,31.515,155.830
C08781=1061.412,189.894,414.949,172.479,31.512,155.830
C08782=1061.406,189.645,414.972,172.477,31.508,155.829
C08783=1061.400,189.396,414.996,172.474,31.506,155.829
C08784=1061.394,189.147,415.020,172.472,31.502,155.828
C08785=1061.389,188.898,415.044,172.470,31.499,155.828
C08786=1061.383,188.649,415.067,172.468,31.497,155.827
C08787=1061.377,188.401,415.091,172.466,31.493,155.827
C08788=1061.372,188.152,415.115,172.464,31.490,155.826
C08789=1061.365,187.903,415.138,172.462,31.487,155.826
C08790=1061.360,187.654,415.162,172.460,31.484,155.825
C08791=1061.354,187.405,415.185,172.457,31.481,155.825
C08792=1061.348,187.157,415.209,172.455,31.478,155.824
C08793=1061.343,186.908,415.233,172.454,31.475,155.824
C08794=1061.337,186.659,415.256,172.452,31.473,155.823
C08795=1061.332,186.409,415.280,172.449,31.469,155.823
C08796=1061.326,186.161,415.304,172.447,31.466,155.822
C08797=1061.320,185.912,415.327,172.445,31.463,155.822
C08798=1061.315,185.664,415.351,172.443,31.460,155.821
C08799=1061.309,185.415,415.374,172.441,31.457,155.821
C08800=1061.303,185.166,415.397,172.439,31.454,155.820
C08801=1061.298,184.917,415.421,172.437,31.451,155.820
C08802=1061.292,184.668,415.444,172.435,31.448,155.819
C08803=1061.286,184.419,415.468,172.433,31.445,155.819
C08804=1061.280,184.171,415.491,172.430,31.442,155.818
C08805=1061.274,183.922,415.514,172.429,31.439,155.818
C08806=1061.268,183.673,415.537,172.427,31.437,155.817
C08807=1061.262,183.424,415.561,172.425,31.434,155.817
C08808=1061.256,183.175,415.584,172.422,31.431,155.817
C08809=1061.250,182.926,415.607,172.420,31.428,155.816
C08810=1061.244,182.678,415.631,172.418,31.425,155.816
C08811=1061.238,182.428,415.654,172.416,31.422,155.815
C08812=1061.232,182.179,415.677,172.414,31.420,155.815
C08813=1061.226,181.931,415.699,172.412,31.416,155.814
C08814=1061.220,181.682,415.723,172.410,31.414,155.814
C08815=1061.214,181.433,415.746,172.408,31.411,155.813
C08816=1061.208,181.185,415.769,172.405,31.408,155.813
C08817=1061.202,180.935,415.792,172.403,31.405,155.812
C08818=1061.196,180.686,415.815,172.402,31.402,155.812
C08819=1061.190,180.437,415.838,172.400,31.399,155.811
C08820=1061.184,180.189,415.862,172.398,31.397,155.811
C08821=1061.179,179.940,415.885,172.395,31.393,155.811
C08822=1061.172,179.691,415.907,172.393,31.391,155.810
C08823=1061.166,179.442,415.930,172.391,31.388,155.810
C08824=1061.160,179.193,415.953,172.390,31.385,155.809
C08825=1061.154,178.944,415.976,172.387,31.382,155.809
C08826=1061.149,178.695,415.999,172.385,31.380,155.808
C08827=1061.143,178.446,416.022,172.383,31.376,155.808
C08828=1061.137,178.198,416.046,172.381,31.374,155.807
C08829=1061.130,177.949,416.068,172.379,31.371,155.807
C08830=1061.125,177.700,416.091,172.378,31.368,155.806
C08831=1061.119,177.452,416.114,172.375,31.365,155.806
C08832=1061.113,177.203,416.137,172.373,31.363,155.806
C08833=1061.107,176.953,416.160,172.371,31.359,155.805
C08834=1061.101,176.704,416.183,172.369,31.357,155.805
C08835=1061.095,176.456,416.205,172.367,31.354,155.804
C08836=1061.089,176.207,416.228,172.365,31.351,155.804
C08837=1061.083,175.958,416.251,172.363,31.348,155.803
C08838=1061.078,175.709,416.274,172.361,31.345,155.803
C08839=1061.072,175.460,416.297,172.359,31.342,155.802
C08840=1061.066,175.211,416.320,172.357,31.340,155.802
C08841=1061.060,174.927,416.345,172.354,31.336,155.801
C08842=1061.053,174.644,416.372,172.353,31.333,155.801
C08843=1061.046,174.360,416.398,172.350,31.330,155.800
C08844=1061.039,174.076,416.424,172.348,31.327,155.800
C08845=1061.033,173.827,416.447,172.346,31.324,155.799
C08846=1061.028,173.578,416.469,172.344,31.321,155.799
C08847=1061.021,173.330,416.492,172.342,31.318,155.798
C08848=1061.015,173.081,416.515,172.340,31.315,155.798
C08849=1061.010,172.832,416.538,172.338,31.312,155.797
C08850=1061.004,172.582,416.560,172.336,31.310,155.797
C08851=1060.999,172.333,416.583,172.334,31.306,155.796
C08852=1060.992,172.085,416.605,172.332,31.304,155.796
C08853=1060.986,171.836,416.628,172.330,31.301,155.796
C08854=1060.981,171.587,416.651,172.328,31.298,155.795
C08855=1060.975,171.338,416.674,172.326,31.295,155.795
C08856=1060.969,171.089,416.696,172.324,31.292,155.794
C08857=1060.964,170.841,416.718,172.322,31.289,155.794
C08858=1060.958,170.592,416.741,172.320,31.287,155.793
C08859=1060.952,170.343,416.764,172.319,31.284,155.793
C08860=1060.947,170.093,416.786,172.317,31.281,155.792
C08861=1060.940,169.845,416.809,172.314,31.278,155.792
C08862=1060.935,169.596,416.832,172.312,31.275,155.791
C08863=1060.929,169.347,416.855,172.310,31.272,155.791
C08864=1060.923,169.097,416.877,172.308,31.270,155.791
C08865=1060.917,168.849,416.899,172.307,31.267,155.790
C08866=1060.911,168.600,416.922,172.305,31.264,155.790
C08867=1060.906,168.352,416.945,172.303,31.261,155.789
C08868=1060.901,168.102,416.967,172.301,31.258,155.789
C08869=1060.894,167.854,416.989,172.299,31.255,155.788
C08870=1060.888,167.605,417.012,172.297,31.253,155.788
C08871=1060.883,167.355,417.035,172.295,31.249,155.787
C08872=1060.877,167.107,417.057,172.293,31.247,155.787
C08873=1060.871,166.857,417.079,172.291,31.244,155.786
C08874=1060.866,166.609,417.102,172.289,31.241,155.786
C08875=1060.860,166.360,417.125,172.287,31.238,155.785
C08876=1060.854,166.111,417.146,172.285,31.236,155.785
C08877=1060.848,165.862,417.169,172.284,31.232,155.784
C08878=1060.843,165.612,417.191,172.282,31.230,155.784
C08879=1060.838,165.364,417.214,172.280,31.227,155.784
C08880=1060.831,165.116,417.236,172.278,31.224,155.783
C08881=1060.826,164.866,417.259,172.276,31.221,155.783
C08882=1060.820,164.617,417.282,172.274,31.218,155.782
C08883=1060.814,164.368,417.303,172.272,31.215,155.782
C08884=1060.809,164.120,417.326,172.270,31.213,155.781
C08885=1060.803,163.870,417.348,172.268,31.209,155.781
C08886=1060.797,163.622,417.370,172.266,31.207,155.780
C08887=1060.792,163.372,417.393,172.264,31.204,155.780
C08888=1060.786,163.124,417.415,172.263,31.201,155.779
C08889=1060.781,162.875,417.437,172.261,31.198,155.779
C08890=1060.775,162.626,417.460,172.259,31.195,155.778
C08891=1060.769,162.376,417.482,172.257,31.192,155.778
C08892=1060.764,162.128,417.505,172.255,31.190,155.778
C08893=1060.758,161.879,417.526,172.253,31.187,155.777
C08894=1060.752,161.630,417.549,172.252,31.184,155.777
C08895=1060.747,161.381,417.571,172.250,31.181,155.776
C08896=1060.741,161.132,417.593,172.248,31.178,155.776
C08897=1060.735,160.883,417.616,172.246,31.175,155.775
C08898=1060.729,160.634,417.637,172.244,31.173,155.775
C08899=1060.723,160.385,417.660,172.242,31.170,155.774
C08900=1060.718,160.137,417.681,172.240,31.167,155.774
C08901=1060.712,159.887,417.703,172.238,31.164,155.774
C08902=1060.705,159.639,417.725,172.236,31.162,155.773
C08903=1060.700,159.389,417.748,172.234,31.159,155.773
C08904=1060.694,159.141,417.769,172.232,31.156,155.772
C08905=1060.687,158.856,417.795,172.231,31.153,155.772
C08906=1060.681,158.572,417.819,172.228,31.150,155.771
C08907=1060.674,158.288,417.844,172.226,31.146,155.771
C08908=1060.668,158.004,417.870,172.224,31.144,155.770
C08909=1060.661,157.755,417.891,172.222,31.141,155.770
C08910=1060.655,157.506,417.913,172.221,31.138,155.769
C08911=1060.650,157.257,417.935,172.219,31.135,155.769
C08912=1060.644,157.008,417.957,172.217,31.133,155.768
C08913=1060.638,156.759,417.979,172.215,31.130,155.768
C08914=1060.632,156.510,418.001,172.213,31.127,155.768
C08915=1060.627,156.261,418.022,172.211,31.124,155.767
C08916=1060.621,156.012,418.044,172.210,31.121,155.767
C08917=1060.615,155.763,418.067,172.207,31.119,155.766
C08918=1060.609,155.514,418.088,172.205,31.116,155.766
C08919=1060.603,155.265,418.110,172.203,31.113,155.765
C08920=1060.597,155.016,418.131,172.201,31.111,155.765
C08921=1060.592,154.767,418.153,172.200,31.108,155.765
C08922=1060.586,154.518,418.175,172.198,31.105,155.764
C08923=1060.580,154.269,418.196,172.196,31.102,155.764
C08924=1060.573,154.020,418.219,172.194,31.100,155.763
C08925=1060.568,153.772,418.240,172.192,31.097,155.763
C08926=1060.562,153.523,418.262,172.190,31.094,155.762
C08927=1060.556,153.273,418.284,172.189,31.092,155.762
C08928=1060.551,153.025,418.305,172.187,31.089,155.762
C08929=1060.544,152.775,418.327,172.185,31.086,155.761
C08930=1060.538,152.526,418.349,172.183,31.083,155.761
C08931=1060.533,152.278,418.370,172.181,31.080,155.760
C08932=1060.527,152.028,418.391,172.180,31.078,155.760
C08933=1060.521,151.779,418.414,172.178,31.075,155.759
C08934=1060.516,151.530,418.435,172.176,31.073,155.759
C08935=1060.509,151.281,418.457,172.174,31.070,155.759
C08936=1060.504,151.033,418.478,172.172,31.067,155.758
C08937=1060.498,150.783,418.499,172.170,31.064,155.758
C08938=1060.492,150.534,418.521,172.169,31.061,155.757
C08939=1060.486,150.286,418.542,172.167,31.059,155.757
C08940=1060.480,150.037,418.564,172.165,31.056,155.756
C08941=1060.474,149.787,418.586,172.163,31.053,155.756
C08942=1060.469,149.539,418.607,172.161,31.051,155.756
C08943=1060.463,149.289,418.629,172.160,31.048,155.755
C08944=1060.457,149.040,418.650,172.158,31.045,155.755
C08945=1060.451,148.791,418.671,172.156,31.042,155.754
C08946=1060.445,148.542,418.693,172.154,31.040,155.754
C08947=1060.440,148.293,418.714,172.152,31.037,155.753
C08948=1060.433,148.044,418.736,172.150,31.034,155.753
C08949=1060.428,147.796,418.757,172.149,31.032,155.752
C08950=1060.422,147.546,418.779,172.147,31.029,155.752
C08951=1060.415,147.297,418.800,172.145,31.026,155.752
C08952=1060.410,147.048,418.821,172.143,31.024,155.751
C08953=1060.404,146.799,418.843,172.141,31.021,155.751
C08954=1060.398,146.550,418.864,172.140,31.018,155.750
C08955=1060.392,146.301,418.885,172.138,31.016,155.750
C08956=1060.386,146.052,418.907,172.137,31.013,155.749
C08957=1060.380,145.803,418.927,172.135,31.010,155.749
C08958=1060.374,145.554,418.949,172.133,31.007,155.749
C08959=1060.368,145.305,418.970,172.131,31.005,155.748
C08960=1060.362,145.056,418.992,172.130,31.002,155.748
C08961=1060.357,144.807,419.012,172.128,30.999,155.747
C08962=1060.351,144.558,419.034,172.126,30.997,155.747
C08963=1060.345,144.309,419.055,172.124,30.994,155.747
C08964=1060.339,144.060,419.076,172.122,30.991,155.746
C08965=1060.333,143.810,419.098,172.121,30.989,155.746
C08966=1060.328,143.562,419.119,172.119,30.986,155.745
C08967=1060.321,143.313,419.140,172.117,30.983,155.745
C08968=1060.316,143.064,419.161,172.115,30.981,155.744
C08969=1060.310,142.779,419.185,172.113,30.978,155.744
C08970=1060.302,142.495,419.209,172.111,30.974,155.743
C08971=1060.296,142.211,419.233,172.109,30.972,155.743
C08972=1060.289,141.927,419.257,172.107,30.968,155.742
C08973=1060.283,141.677,419.278,172.105,30.966,155.742
C08974=1060.277,141.428,419.300,172.103,30.963,155.742
C08975=1060.272,141.178,419.321,172.102,30.960,155.741
C08976=1060.266,140.930,419.342,172.100,30.958,155.741
C08977=1060.260,140.681,419.363,172.098,30.955,155.740
C08978=1060.254,140.432,419.383,172.096,30.952,155.740
C08979=1060.248,140.183,419.405,172.094,30.950,155.740
C08980=1060.242,139.934,419.426,172.094,30.947,155.739
C08981=1060.236,139.684,419.447,172.092,30.945,155.739
C08982=1060.231,139.435,419.468,172.090,30.942,155.738
C08983=1060.224,139.186,419.489,172.088,30.939,155.738
C08984=1060.219,138.937,419.509,172.086,30.936,155.737
C08985=1060.213,138.688,419.531,172.084,30.933,155.737
C08986=1060.207,138.439,419.551,172.083,30.931,155.736
C08987=1060.201,138.190,419.573,172.081,30.928,155.736
C08988=1060.195,137.941,419.593,172.079,30.925,155.736
C08989=1060.190,137.692,419.614,172.077,30.923,155.735
C08990=1060.183,137.443,419.635,172.075,30.920,155.735
C08991=1060.178,137.194,419.656,172.074,30.917,155.734
C08992=1060.172,136.945,419.677,172.072,30.915,155.734
C08993=1060.165,136.696,419.698,172.070,30.912,155.734
C08994=1060.160,136.446,419.719,172.069,30.910,155.733
C08995=1060.154,136.198,419.739,172.067,30.907,155.733
C08996=1060.147,135.948,419.760,172.066,30.904,155.732
C08997=1060.142,135.699,419.781,172.064,30.902,155.732
C08998=1060.136,135.451,419.801,172.062,30.899,155.732
C08999=1060.130,135.201,419.822,172.060,30.896,155.731
C09000=1060.125,134.952,419.843,172.058,30.894,155.731
C09001=1060.118,134.703,419.864,172.057,30.891,155.730
C09002=1060.113,134.454,419.884,172.055,30.888,155.730
C09003=1060.107,134.205,419.904,172.053,30.886,155.729
C09004=1060.100,133.956,419.926,172.051,30.883,155.729
C09005=1060.095,133.707,419.947,172.049,30.880,155.729
C09006=1060.089,133.458,419.967,172.048,30.878,155.728
C09007=1060.083,133.209,419.988,172.047,30.875,155.728
C09008=1060.078,132.960,420.009,172.045,30.872,155.727
C09009=1060.071,132.710,420.029,172.043,30.870,155.727
C09010=1060.066,132.461,420.050,172.041,30.867,155.727
C09011=1060.060,132.213,420.070,172.039,30.864,155.726
C09012=1060.054,131.963,420.091,172.038,30.862,155.726
C09013=1060.048,131.714,420.112,172.036,30.859,155.725
C09014=1060.042,131.465,420.132,172.034,30.856,155.725
C09015=1060.036,131.216,420.153,172.032,30.854,155.724
C09016=1060.030,130.967,420.173,172.031,30.851,155.724
C09017=1060.024,130.718,420.194,172.030,30.849,155.724
C09018=1060.018,130.469,420.214,172.028,30.847,155.723
C09019=1060.012,130.220,420.234,172.026,30.844,155.723
C09020=1060.006,129.971,420.255,172.024,30.841,155.722
C09021=1060.000,129.722,420.275,172.022,30.839,155.722
C09022=1059.994,129.472,420.296,172.021,30.836,155.722
C09023=1059.988,129.223,420.316,172.019,30.833,155.721
C09024=1059.982,128.975,420.336,172.017,30.831,155.721
C09025=1059.976,128.725,420.357,172.015,30.828,155.720
C09026=1059.970,128.476,420.377,172.014,30.826,155.720
C09027=1059.964,128.227,420.397,172.013,30.823,155.720
C09028=1059.958,127.978,420.418,172.011,30.821,155.719
C09029=1059.952,127.729,420.438,172.009,30.818,155.719
C09030=1059.946,127.480,420.458,172.007,30.815,155.718
C09031=1059.940,127.231,420.479,172.005,30.813,155.718
C09032=1059.934,126.982,420.499,172.004,30.810,155.718
C09033=1059.927,126.697,420.523,172.002,30.807,155.717
C09034=1059.920,126.413,420.545,172.000,30.804,155.717
C09035=1059.913,126.127,420.569,171.998,30.801,155.716
C09036=1059.906,125.843,420.592,171.996,30.798,155.716
C09037=1059.901,125.594,420.612,171.995,30.795,155.715
C09038=1059.895,125.345,420.632,171.993,30.793,155.715
C09039=1059.888,125.096,420.652,171.991,30.790,155.714
C09040=1059.883,124.846,420.673,171.989,30.788,155.714
C09041=1059.877,124.598,420.693,171.987,30.785,155.714
C09042=1059.871,124.349,420.713,171.986,30.783,155.713
C09043=1059.864,124.099,420.733,171.985,30.780,155.713
C09044=1059.859,123.850,420.754,171.983,30.777,155.713
C09045=1059.853,123.601,420.774,171.981,30.775,155.712
C09046=1059.847,123.353,420.794,171.979,30.772,155.712
C09047=1059.841,123.103,420.815,171.978,30.769,155.711
C09048=1059.835,122.854,420.835,171.976,30.767,155.711
C09049=1059.829,122.605,420.855,171.974,30.764,155.710
C09050=1059.823,122.356,420.875,171.973,30.762,155.710
C09051=1059.818,122.106,420.895,171.971,30.759,155.710
C09052=1059.812,121.857,420.915,171.970,30.756,155.709
C09053=1059.806,121.608,420.935,171.968,30.754,155.709
C09054=1059.800,121.359,420.955,171.966,30.751,155.708
C09055=1059.795,121.110,420.975,171.964,30.748,155.708
C09056=1059.788,120.861,420.995,171.962,30.746,155.708
C09057=1059.782,120.612,421.015,171.962,30.743,155.707
C09058=1059.776,120.363,421.035,171.960,30.741,155.707
C09059=1059.771,120.113,421.055,171.958,30.738,155.706
C09060=1059.765,119.865,421.075,171.956,30.736,155.706
C09061=1059.759,119.615,421.096,171.954,30.733,155.706
C09062=1059.753,119.366,421.115,171.953,30.730,155.705
C09063=1059.747,119.117,421.136,171.952,30.728,155.705
C09064=1059.742,118.868,421.155,171.950,30.725,155.704
C09065=1059.736,118.619,421.175,171.948,30.722,155.704
C09066=1059.730,118.370,421.195,171.946,30.720,155.704
C09067=1059.724,118.121,421.216,171.945,30.717,155.703
C09068=1059.718,117.871,421.235,171.943,30.714,155.703
C09069=1059.712,117.622,421.255,171.942,30.712,155.702
C09070=1059.706,117.373,421.275,171.940,30.709,155.702
C09071=1059.700,117.124,421.295,171.938,30.706,155.701
C09072=1059.695,116.875,421.315,171.937,30.704,155.701
C09073=1059.689,116.626,421.335,171.935,30.701,155.701
C09074=1059.683,116.377,421.355,171.933,30.698,155.700
C09075=1059.677,116.128,421.375,171.932,30.696,155.700
C09076=1059.672,115.878,421.395,171.930,30.693,155.699
C09077=1059.666,115.629,421.415,171.929,30.691,155.699
C09078=1059.660,115.380,421.435,171.927,30.688,155.699
C09079=1059.654,115.131,421.454,171.925,30.685,155.698
C09080=1059.648,114.882,421.474,171.924,30.683,155.698
C09081=1059.643,114.632,421.494,171.923,30.680,155.697
C09082=1059.637,114.383,421.514,171.921,30.677,155.697
C09083=1059.631,114.134,421.534,171.919,30.675,155.696
C09084=1059.625,113.885,421.553,171.917,30.672,155.696
C09085=1059.619,113.636,421.573,171.915,30.669,155.696
C09086=1059.614,113.387,421.592,171.915,30.667,155.695
C09087=1059.607,113.137,421.613,171.913,30.664,155.695
C09088=1059.601,112.888,421.633,171.911,30.661,155.694
C09089=1059.595,112.639,421.652,171.909,30.659,155.694
C09090=1059.589,112.390,421.672,171.907,30.656,155.694
C09091=1059.584,112.141,421.691,171.906,30.654,155.693
C09092=1059.578,111.892,421.711,171.905,30.651,155.693
C09093=1059.572,111.643,421.730,171.903,30.649,155.692
C09094=1059.566,111.394,421.750,171.901,30.646,155.692
C09095=1059.560,111.144,421.770,171.899,30.643,155.692
C09096=1059.554,110.896,421.789,171.898,30.641,155.691
C09097=1059.547,110.610,421.812,171.896,30.638,155.691
C09098=1059.540,110.326,421.834,171.894,30.635,155.690
C09099=1059.533,110.041,421.856,171.892,30.632,155.690
C09100=1059.527,109.756,421.878,171.891,30.629,155.689
C09101=1059.521,109.507,421.898,171.889,30.627,155.689
C09102=1059.514,109.258,421.917,171.887,30.624,155.689
C09103=1059.508,109.009,421.937,171.886,30.621,155.688
